# B&R Automation Studio project mappFramework (part 3)

#### AsLoggerFile.c
```c
/********************************************************************
 * COPYRIGHT -- Bernecker + Rainer
 ********************************************************************
 * Library: AsLogger
 * File: AsLoggerFile.c
 * Author: buchananw
 * Created: August 21, 2009
 *******************************************************************/

#include <bur/plctypes.h>
#include <LoggingLib.h>
#include <string.h>
#include <stdbool.h>
#include "AsLoggerInternal.h"

#ifdef __DEBUG_LOGGING_LIBRARY__
#define transit(x, _state)                                          \
{                                                                   \
    x = _state;                                                     \
    logDebug("AsLoggerFile", "changing to state " #_state, NULL);   \
}
#else

#define transit(x, _state)                                          \
{                                                                   \
    x = _state;                                                     \
}

#endif

#define disableAllFunctionBlocks                \
inst->internal.FileOpen_0.enable    = false;    \
inst->internal.FileCreate_0.enable  = false;    \
inst->internal.FileWrite_0.enable   = false;    \
inst->internal.FileCopy_0.enable    = false;    \
inst->internal.FileClose_0.enable   = false;    \
inst->internal.FileDelete_0.enable  = false;

#define incrementFileNumber(x) x = (x+1) % inst->maxFiles
#define decrementFileNumber(x) x = (x > 0) ? x - 1 : inst->maxFiles - 1

void AsLoggerFile(struct AsLoggerFile* inst)
{
    LogStore_typ* logStore;
    UDINT arguments[LOGGING_MAX_ARGUMENTS];
    USINT i;

    if (inst == NULL)
    {
        logError("AsLoggerFile", "AsLoggerFile called with NULL instance", (UDINT)NULL);
        return;
    }
    logStore = getLogStore();

    if (logStore == NULL)
    {
        transit(inst->internal.state, AS_FILE_LOGGER_STATE_ERROR);
#ifdef __DEBUG_LOGGING_LIBRARY__
        logDebug("AsLoggerFile", "logStore is NULL", NULL);
        logDebug("AsLoggerFile", "changing to ERROR state", NULL);
#endif
        inst->status = ASLOGGER_INTERNAL_ERROR;
        return;
    }

    switch(inst->internal.state)
    {
        case AS_FILE_LOGGER_STATE_W_ENABLE:
            if (inst->enable != true)
            {
                inst->status = ERR_FUB_ENABLE_FALSE;
                return;
            }

            if (strcmp(inst->device, "") == true)
            {
                logError("AsLoggerFile", "device name empty", (UDINT)NULL);
                inst->status = ASLOGGER_ILLEGAL_DEVICENAME;
                return;
            }
            if (strcmp(inst->fileName, "") == true)
            {
                logError("AsLoggerFile", "file name empty", (UDINT)NULL);
                inst->status = ASLOGGER_ILLEGAL_FILENAME;
                return;
            }

            inst->internal.fileNumber = (inst->maxFiles > 1) ? inst->maxFiles - 1 : 0;
            if (inst->internal.fileNumber <= 1)
            {
                snprintf2(inst->internal.tempFileName, (sizeof(inst->internal.tempFileName) / sizeof(inst->internal.tempFileName[0])) - 1, "%s.%s", inst->fileName, inst->fileExtension);
                inst->internal.FileDelete_0.pDevice = (UDINT)&inst->device;
                inst->internal.FileDelete_0.pName = (UDINT)&inst->internal.tempFileName;
                inst->internal.FileDelete_0.enable = true;
                transit(inst->internal.state, AS_FILE_LOGGER_STATE_DELETE_OLD);
            }
            else
            {
                snprintf2(inst->internal.newFileName, (sizeof(inst->internal.newFileName) / sizeof(inst->internal.newFileName[0])) - 1, "%s%d.%s", inst->fileName, inst->internal.fileNumber, inst->fileExtension);
                snprintf2(inst->internal.oldFileName, (sizeof(inst->internal.oldFileName) / sizeof(inst->internal.oldFileName[0])) - 1, "%s%d.%s", inst->fileName, --inst->internal.fileNumber, inst->fileExtension);

                inst->internal.FileCopy_0.enable = true;
                inst->internal.FileCopy_0.option = fiOVERWRITE;
                inst->internal.FileCopy_0.pSrc = (UDINT)&inst->internal.oldFileName;
                inst->internal.FileCopy_0.pSrcDev = (UDINT)&inst->device;
                inst->internal.FileCopy_0.pDest = (UDINT)&inst->internal.newFileName;
                inst->internal.FileCopy_0.pDestDev = (UDINT)&inst->device;
                transit(inst->internal.state, AS_FILE_LOGGER_STATE_MOVE_FILES);
            }
        break;

        case AS_FILE_LOGGER_STATE_MOVE_FILES:
            switch (inst->internal.FileCopy_0.status)
            {
                case 0:
                case fiERR_FILE_NOT_FOUND:
                    inst->internal.FileCopy_0.enable = false;
                    if (inst->internal.fileNumber == 0)
                    {
                        snprintf2(inst->internal.tempFileName, (sizeof(inst->internal.tempFileName) / sizeof(inst->internal.tempFileName[0])) - 1, "%s.%s", inst->fileName, inst->fileExtension);
                        inst->internal.FileDelete_0.pDevice = (UDINT)&inst->device;
                        inst->internal.FileDelete_0.pName = (UDINT)&inst->internal.tempFileName;
                        inst->internal.FileDelete_0.enable = true;
                        transit(inst->internal.state, AS_FILE_LOGGER_STATE_DELETE_OLD);
                    }
                    else
                    {
                        strcpy((char*)&inst->internal.newFileName, (char*)&inst->internal.oldFileName);

                        if (inst->internal.fileNumber <= 1)
                        {
                            snprintf2(inst->internal.oldFileName, (sizeof(inst->internal.oldFileName) / sizeof(inst->internal.oldFileName[0])) - 1, "%s.%s", inst->fileName, inst->fileExtension);
                            inst->internal.fileNumber--;
                        }
                        else
                        {
                            snprintf2(inst->internal.oldFileName, (sizeof(inst->internal.oldFileName) / sizeof(inst->internal.oldFileName[0])) - 1, "%s%d.%s", inst->fileName, --inst->internal.fileNumber, inst->fileExtension);
                        }
                        inst->internal.FileCopy_0.option = fiOVERWRITE;
                        inst->internal.FileCopy_0.pSrc = (UDINT)&inst->internal.oldFileName;
                        inst->internal.FileCopy_0.pSrcDev = (UDINT)&inst->device;
                        inst->internal.FileCopy_0.pDest = (UDINT)&inst->internal.newFileName;
                        inst->internal.FileCopy_0.pDestDev = (UDINT)&inst->device;
                        /* no state transition here. */
                    }
                break;

                case ERR_FUB_ENABLE_FALSE:
                    inst->internal.FileCopy_0.enable = true;
                break;

                case ERR_FUB_BUSY:
                break;

                default:
                    disableAllFunctionBlocks;
#ifdef __DEBUG_LOGGING_LIBRARY__
                    //snprintf2(logString, (sizeof(logString) / sizeof(logString[0])) - 1, "old file name %s", inst->internal.oldFileName);
                    //snprintf2(logString, (sizeof(logString) / sizeof(logString[0])) - 1, "new file name %s", inst->internal.newFileName);
                    //logDebug("AsLoggerFile", logString);
                    arguments[0] = (UDINT)inst->internal.oldFileName;
                    arguments[1] = (UDINT)inst->internal.newFileName;
                    logDebug("AsLoggerFile", "old file name is %s, new file name is %s", (UDINT)&arguments);

#endif
                    //snprintf2(logString, (sizeof(logString) / sizeof(logString[0])) - 1, "file copy error %d", inst->internal.FileCopy_0.status);
                    arguments[0] = (UDINT)&inst->internal.FileCopy_0.status;
                    logDebug("AsLoggerFile", "file copy error %d", (UDINT)&arguments);
                    logDebug("AsLoggerFile", "changing to ERROR state", (UDINT)NULL);

                    transit(inst->internal.state, AS_FILE_LOGGER_STATE_ERROR);
                break;
            }
        break;

        case AS_FILE_LOGGER_STATE_DELETE_OLD:

            switch (inst->internal.FileDelete_0.status)
            {
                case 0:
                case fiERR_FILE_NOT_FOUND:
                    inst->internal.FileDelete_0.enable = false;
                    inst->internal.FileCreate_0.pDevice = (UDINT)&inst->device;
                    snprintf2(inst->internal.tempFileName, (sizeof(inst->internal.tempFileName) / sizeof(inst->internal.tempFileName[0]))- 1, "%s.%s", inst->fileName, inst->fileExtension);
                    inst->internal.FileCreate_0.pFile = (UDINT)&inst->internal.tempFileName;
                    inst->internal.FileCreate_0.enable = true;
                    transit(inst->internal.state, AS_FILE_LOGGER_STATE_CREATE_FILE);
                break;

                case ERR_FUB_ENABLE_FALSE:
                    inst->internal.FileDelete_0.enable = true;
                break;

                case ERR_FUB_BUSY:
                break;

                default:
                    disableAllFunctionBlocks;
                    //snprintf2(logString, (sizeof(logString) / sizeof(logString[0])) - 1, "file delete error %d", inst->internal.FileDelete_0.status);
                    arguments[0] = (UDINT)&inst->internal.FileDelete_0.status;
                    logDebug("AsLoggerFile", "file delete error %d", (UDINT)&arguments);
                    logDebug("AsLoggerFile", "changing to ERROR state", (UDINT)NULL);
                    transit(inst->internal.state, AS_FILE_LOGGER_STATE_ERROR);
                break;
            }
        break;

        case AS_FILE_LOGGER_STATE_CREATE_FILE:
            switch (inst->internal.FileCreate_0.status)
            {
                case 0:
                    inst->internal.FileCreate_0.enable = false;
                    inst->internal.FileClose_0.ident = inst->internal.FileCreate_0.ident;
                    inst->internal.FileClose_0.enable = true;
                    inst->internal.fileOffset = 0;
                    inst->internal.writeBufferUsed = 0;
                    transit(inst->internal.state, AS_FILE_LOGGER_STATE_CLOSE);
                break;

                case ERR_FUB_ENABLE_FALSE:
                    inst->internal.FileCreate_0.enable = true;
                break;

                case ERR_FUB_BUSY:
                break;

                default:
                    disableAllFunctionBlocks;
                    //snprintf2(logString, (sizeof(logString) / sizeof(logString[0])) - 1, "file create error %d", inst->internal.FileCreate_0.status);
                    arguments[0] = (UDINT)&inst->internal.FileCreate_0.status;
                    logDebug("AsLoggerFile", "file create error %d", (UDINT)&arguments);
                    logDebug("AsLoggerFile", "changing to ERROR state", (UDINT)NULL);
                    logDebug("AsLoggerFile", inst->internal.tempFileName, (UDINT)NULL);
                    transit(inst->internal.state, AS_FILE_LOGGER_STATE_ERROR);
                    inst->status = inst->internal.FileCreate_0.status;
            }
        break;

        case AS_FILE_LOGGER_STATE_MARSHALL:
            memset(&inst->internal.writeBuffer, 0, sizeof(inst->internal.writeBuffer));
            inst->internal.writeBufferUsed = 0;

            for (i=inst->internal.outputIndex; i != logStore->inputIndex; incrementIndex(i))
            {
                if (logStore->messages[i].level >= inst->level)
                {
                    memset(inst->internal.tempString, 0, sizeof(inst->internal.tempString));
                    marchallLogMessageForFile(&logStore->messages[i], inst->delimiter, inst->internal.tempString, sizeof(inst->internal.tempString) / sizeof(inst->internal.tempString[0]));
                    if ((strlen(inst->internal.tempString) + inst->internal.writeBufferUsed) >= sizeof(inst->internal.writeBuffer))
                    {
                        snprintf2(inst->internal.tempFileName, (sizeof(inst->internal.tempFileName) / sizeof(inst->internal.tempFileName[0])) - 1, "%s.%s", inst->fileName, inst->fileExtension);
                        inst->internal.FileOpen_0.enable = true;
                        inst->internal.FileOpen_0.mode = fiREAD_WRITE;
                        inst->internal.FileOpen_0.pDevice = (UDINT)&inst->device;
                        inst->internal.FileOpen_0.pFile = (UDINT)&inst->internal.tempFileName;
                        transit(inst->internal.state, AS_FILE_LOGGER_STATE_OPEN);
                        return;
                    }
                    addStringToBuffer((char*)&inst->internal.writeBuffer, &inst->internal.writeBufferUsed, inst->internal.tempString);
                }
                incrementIndex(inst->internal.outputIndex);
            }
            if (inst->internal.writeBufferUsed > 0)
            {
                snprintf2(inst->internal.tempFileName, (sizeof(inst->internal.tempFileName) / sizeof(inst->internal.tempFileName[0]))- 1, "%s.%s", inst->fileName, inst->fileExtension);
                inst->internal.FileOpen_0.enable = true;
                inst->internal.FileOpen_0.mode = fiREAD_WRITE;
                inst->internal.FileOpen_0.pDevice = (UDINT)&inst->device;
                inst->internal.FileOpen_0.pFile = (UDINT)&inst->internal.tempFileName;
                transit(inst->internal.state, AS_FILE_LOGGER_STATE_OPEN);
            }
        break;

        case AS_FILE_LOGGER_STATE_OPEN:
            switch (inst->internal.FileOpen_0.status)
            {
                case 0:
                    inst->internal.FileOpen_0.enable = false;

                    inst->internal.FileWrite_0.enable = true;
                    inst->internal.FileWrite_0.ident = inst->internal.FileOpen_0.ident;
                    inst->internal.FileWrite_0.len = inst->internal.writeBufferUsed;
                    inst->internal.FileWrite_0.offset = inst->internal.fileOffset;
                    inst->internal.FileWrite_0.pSrc = (UDINT)inst->internal.writeBuffer;
                    transit(inst->internal.state, AS_FILE_LOGGER_STATE_WRITE);
                break;

                case ERR_FUB_ENABLE_FALSE:
                    inst->internal.FileOpen_0.enable = true;
                break;

                case ERR_FUB_BUSY:
                break;

                default:
                    disableAllFunctionBlocks;
                    //snprintf2(logString, (sizeof(logString) / sizeof(logString[0])) - 1, "file open error %d", inst->internal.FileOpen_0.status);
                    arguments[0] = (UDINT)&inst->internal.FileOpen_0.status;
                    logDebug("AsLoggerFile", "file open error %d", (UDINT)&arguments);
                    logDebug("AsLoggerFile", "changing to ERROR state", (UDINT)NULL);
                    logDebug("AsLoggerFile", inst->internal.tempFileName, (UDINT)NULL);
                    transit(inst->internal.state, AS_FILE_LOGGER_STATE_ERROR);
                    inst->status = inst->internal.FileOpen_0.status;
            }
        break;

        case AS_FILE_LOGGER_STATE_WRITE:
            switch (inst->internal.FileWrite_0.status)
            {
                case 0:
                    inst->internal.FileWrite_0.enable = false;
                    inst->internal.fileOffset += inst->internal.writeBufferUsed;
                    inst->internal.FileClose_0.enable = true;
                    inst->internal.FileClose_0.ident = inst->internal.FileWrite_0.ident;
                    transit(inst->internal.state, AS_FILE_LOGGER_STATE_CLOSE);
                break;

                case ERR_FUB_ENABLE_FALSE:
                    inst->internal.FileWrite_0.enable = true;
                break;

                case ERR_FUB_BUSY:
                break;

                default:
                    disableAllFunctionBlocks;
                    //snprintf2(logString, (sizeof(logString) / sizeof(logString[0])) - 1, "file write error %d", inst->internal.FileWrite_0.status);
                    arguments[0] = (UDINT)&inst->internal.FileWrite_0.status;
                    logDebug("AsLoggerFile", "file write error %d", (UDINT)&arguments);
                    logDebug("AsLoggerFile", "changing to ERROR state", (UDINT)NULL);
                    logDebug("AsLoggerFile", inst->internal.tempFileName, (UDINT)NULL);
                    transit(inst->internal.state, AS_FILE_LOGGER_STATE_ERROR);
                    inst->status = inst->internal.FileWrite_0.status;
            }
        break;

        case AS_FILE_LOGGER_STATE_CLOSE:
            switch (inst->internal.FileClose_0.status)
            {
                case 0:
                    inst->internal.FileClose_0.enable = false;
                    if (inst->internal.fileOffset >= inst->maxFileSize)
                    {
                        inst->internal.fileNumber = (inst->maxFiles > 1) ? inst->maxFiles - 1 : 0;
                        if (inst->internal.fileNumber <= 1)
                        {
                            snprintf2(inst->internal.tempFileName, (sizeof(inst->internal.tempFileName) / sizeof(inst->internal.tempFileName[0])) - 1, "%s.%s", inst->fileName, inst->fileExtension);
                            inst->internal.FileDelete_0.pDevice = (UDINT)&inst->device;
                            inst->internal.FileDelete_0.pName = (UDINT)&inst->internal.tempFileName;
                            inst->internal.FileDelete_0.enable = true;
                            transit(inst->internal.state, AS_FILE_LOGGER_STATE_DELETE_OLD);
                        }
                        else
                        {
                            snprintf2(inst->internal.newFileName, (sizeof(inst->internal.newFileName) / sizeof(inst->internal.newFileName[0])) - 1, "%s%d.%s", inst->fileName, inst->internal.fileNumber, inst->fileExtension);
                            snprintf2(inst->internal.oldFileName, (sizeof(inst->internal.oldFileName) / sizeof(inst->internal.oldFileName[0])) - 1, "%s%d.%s", inst->fileName, --inst->internal.fileNumber, inst->fileExtension);

                            inst->internal.FileCopy_0.enable = true;
                            inst->internal.FileCopy_0.option = fiOVERWRITE;
                            inst->internal.FileCopy_0.pSrc = (UDINT)&inst->internal.oldFileName;
                            inst->internal.FileCopy_0.pSrcDev = (UDINT)&inst->device;
                            inst->internal.FileCopy_0.pDest = (UDINT)&inst->internal.newFileName;
                            inst->internal.FileCopy_0.pDestDev = (UDINT)&inst->device;
                            transit(inst->internal.state, AS_FILE_LOGGER_STATE_MOVE_FILES);
                        }
                    }
                    else
                    {
                        inst->internal.writeBufferUsed = 0;
                        transit(inst->internal.state, AS_FILE_LOGGER_STATE_MARSHALL);
                    }
                break;

                case ERR_FUB_ENABLE_FALSE:
                    inst->internal.FileClose_0.enable = true;
                break;

                case ERR_FUB_BUSY:
                break;

                default:
                    disableAllFunctionBlocks;
                    //snprintf2(logString, (sizeof(logString) / sizeof(logString[0])) - 1, "file close error %d", inst->internal.FileClose_0.status);
                    arguments[0] = (UDINT)&inst->internal.FileClose_0.status;
                    logDebug("AsLoggerFile", "file close error %d", (UDINT)&arguments);
                    logDebug("AsLoggerFile", "changing to ERROR state", (UDINT)NULL);
                    logDebug("AsLoggerFile", inst->internal.tempFileName, (UDINT)NULL);
                    transit(inst->internal.state, AS_FILE_LOGGER_STATE_ERROR);
                    inst->status = inst->internal.FileClose_0.status;
            }
        break;

        case AS_FILE_LOGGER_STATE_ERROR:
            if (inst->enable != true)
            {
                transit(inst->internal.state, 0);
            }
        break;

        default:
        break;
    }

    if (inst->internal.state != AS_FILE_LOGGER_STATE_ERROR)
        inst->status = ERR_FUB_BUSY;

    FileOpen(&inst->internal.FileOpen_0);
    FileWrite(&inst->internal.FileWrite_0);
    FileClose(&inst->internal.FileClose_0);
    FileCreate(&inst->internal.FileCreate_0);
    FileCopy(&inst->internal.FileCopy_0);
    FileDelete(&inst->internal.FileDelete_0);
}

void marchallLogMessageForFile(LogMessage_typ* message, char* delimiter, char* tempString, UDINT sizeOfTempString)
{
    DTStructure timeStamp;
    char level[6];

    if ((message == NULL) || (delimiter == NULL) || (tempString == NULL))
        return;

    DT_TO_DTStructure(message->timeStamp, (UDINT)&timeStamp);
    timeStamp.millisec = message->timeStampMilliseconds;

    memset(&level, 0, sizeof(level));
    switch(message->level)
    {
        case LOG_LEVEL_DEBUG:
            strcpy(level, "DEBUG");
        break;
        case LOG_LEVEL_INFO:
            strcpy(level, "INFO");
        break;
        case LOG_LEVEL_WARN:
            strcpy(level, "WARN");
        break;
        case LOG_LEVEL_ERROR:
            strcpy(level, "ERROR");
        break;
        case LOG_LEVEL_FATAL:
            strcpy(level, "FATAL");
        break;
    }

    snprintf2(tempString, sizeOfTempString - 1, "%04d/%02d/%02d %02d:%02d:%02d.%03d%s %s%s %s%s %s\r\n", timeStamp.year, timeStamp.month, timeStamp.day, \
                    timeStamp.hour, timeStamp.minute, timeStamp.second, timeStamp.millisec, delimiter, \
                    level, delimiter, \
                    message->name, delimiter, \
                    message->message);
}

void addStringToBuffer(char* buffer, UINT* bufferPos, char* newMessage)
{
    if ((buffer == NULL) || (bufferPos == NULL) || (newMessage == NULL))
        return;

    memcpy(buffer + *bufferPos, newMessage, strlen(newMessage));
    *bufferPos = *bufferPos + strlen(newMessage);
}
```

#### AsLoggerLogBook.c
```c
/********************************************************************
 * COPYRIGHT -- Bernecker + Rainer
 ********************************************************************
 * Library: LoggingLib
 * File: AsLoggerLogBook.c
 * Author: buchananw
 * Created: April 19, 2010
 *******************************************************************/

#include <bur/plctypes.h>
#include <LoggingLib.h>
#include <string.h>
#include <stdbool.h>
#include "AsLoggerInternal.h"

#define LOGBOOK_ERROR_STATE 255

#ifdef __DEBUG_LOGGING_LIBRARY__
#define transit(x, y)                                        \
{                                                            \
    x->internal.state = y;                                   \
    logDebug("AsLoggerFile", "changing to state " #y, NULL); \
}
#else
#define transit(x, y)                                        \
{                                                            \
    x->internal.state = y;                                   \
}
#endif

#define incrementFileNumber(x) x = (x+1) % inst->internal.maxFiles
#define decrementFileNumber(x) x = (x > 0) ? x - 1 : inst->internal.maxFiles - 1

void AsLoggerLogBook(struct AsLoggerLogBook* inst)
{
    LogStore_typ* logStore;
#ifdef __DEBUG_LOGGING_LIBRARY__
    UDINT arguments[LOGGING_MAX_ARGUMENTS];
#endif

    if (inst == NULL)
    {
        logError("AsLoggerLogBook", "AsLoggerLogBook called with NULL instance", NULL);
        return;
    }
    logStore = getLogStore();

    if (logStore == NULL)
    {
#ifdef __DEBUG_LOGGING_LIBRARY__
        logDebug("AsLoggerLogBook", "logStore is NULL", NULL);
#endif
        inst->status = ASLOGGER_INTERNAL_ERROR;
        return;
    }

    if (inst->internal.outputIndexRegistered != true)
    {
        addNewOutputIndex(&inst->internal.outputIndex);
        inst->internal.outputIndexRegistered = true;
    }

    while ((inst->internal.outputIndex != logStore->inputIndex) && (logStore->messages[inst->internal.outputIndex].level < inst->level))
    {
        incrementIndex(inst->internal.outputIndex);
    }

    if (inst->internal.outputIndex != logStore->inputIndex)
    {
        if (inst->internal.ArEventLogWrite_0.Ident == 0)
        {
            inst->internal.ArEventLogGetIdent_0.Execute = true;
            strcpy(inst->internal.ArEventLogGetIdent_0.Name, "$arlogusr");
            ArEventLogGetIdent(&inst->internal.ArEventLogGetIdent_0);
            if (inst->internal.ArEventLogGetIdent_0.StatusID == 0)
                inst->internal.ArEventLogWrite_0.Ident = inst->internal.ArEventLogGetIdent_0.Ident;
        }
        else
        {
            USINT _logBuffer[MAX_MESSAGE_LENGTH + MAX_NAME_LENGTH + 10];
            char _tempString[MAX_MESSAGE_LENGTH + MAX_NAME_LENGTH + 2];

            memset(&_logBuffer, 0, sizeof(_logBuffer));
            inst->internal.ArEventLogWrite_0.Execute = true;
            inst->internal.ArEventLogWrite_0.EventID = ArEventLogMakeEventID(convertToArLogLevel(&(logStore->messages[inst->internal.outputIndex])), 0, 0);
            inst->internal.ArEventLogWrite_0.OriginRecordID = 0;
            snprintf2(_tempString, (sizeof(_tempString) / sizeof(_tempString)) - 1, "%s: %s", logStore->messages[inst->internal.outputIndex].name, logStore->messages[inst->internal.outputIndex].message);
            ArEventLogAddDataInit((UDINT)&_logBuffer, sizeof(_logBuffer), arEVENTLOG_ADDFORMAT_CODED);
            ArEventLogAddDataString((UDINT)&_logBuffer, sizeof(_logBuffer), (UDINT)&_tempString);
            inst->internal.ArEventLogWrite_0.AddData = (UDINT)&_logBuffer;
            inst->internal.ArEventLogWrite_0.AddDataFormat = arEVENTLOG_ADDFORMAT_CODED;
            inst->internal.ArEventLogWrite_0.AddDataSize = sizeof(_logBuffer);

            ArEventLogWrite(&inst->internal.ArEventLogWrite_0);
            if (inst->internal.ArEventLogWrite_0.StatusID == 0)
            {
                incrementIndex(inst->internal.outputIndex);

            }
#ifdef __DEBUG_LOGGING_LIBRARY__
            else
            {
                //snprintf2(logString, (sizeof(logString) / sizeof(logString[0])) - 1, "AR log write error %d", inst->internal.AsArLogWrite_0.status);
                arguments[0] = (UDINT)&inst->internal.ArEventLogWrite_0.StatusID;
                logDebug("AsLoggerLogBook", "AR log write error %d", (UDINT)&arguments);
                inst->status = inst->internal.ArEventLogWrite_0.StatusID;
            }
#endif
            inst->internal.ArEventLogWrite_0.Execute = false;
            ArEventLogWrite(&inst->internal.ArEventLogWrite_0);

        }

    }
}

USINT convertToArLogLevel(LogMessage_typ* message)
{
    if (message == NULL)
        return arEVENTLOG_SEVERITY_INFO;

    switch(message->level)
    {
        case LOG_LEVEL_DEBUG:
        case LOG_LEVEL_INFO:
            return arEVENTLOG_SEVERITY_INFO;
        break;
        case LOG_LEVEL_WARN:
            return arEVENTLOG_SEVERITY_WARNING;
        break;
        case LOG_LEVEL_ERROR:
        case LOG_LEVEL_FATAL:
            return arEVENTLOG_SEVERITY_ERROR;
            return arEVENTLOG_SEVERITY_ERROR;
        break;
    }
    return arEVENTLOG_SEVERITY_ERROR;
}
```


### Package Logical/Infrastructure - Package for Machine Infrastructure

### mappFrameworkGlobal.var - Global variables for the mapp Framework
```iecst
(*Recipe*)
VAR CONSTANT
	MACH_CONFIG_CATEGORY_INDEX : USINT := 1; (*Recipe category index for machine config*)
	PARAMETERS_CATEGORY_INDEX : USINT := 0; (*Recipe category index for machine parameters*)
	PARAMETERS_CATEGORY : STRING[10] := 'Parameters'; (*Recipe category for runtime parameters*)
	MACHINE_CONFIGURATION_CATEGORY : STRING[30] := 'Machine Configuration'; (*Recipe category for machine configuration settings*)
	DEFAULT_PARAMETERS : STRING[20] := 'Default'; (*Default parameters recipe file name*)
	PARAMETERS_FILE_EXTENSION : STRING[10] := '.par'; (*File extension for parameter recipe files*)
	DEFAULT_MACHINE_CONFIGURATION : STRING[20] := 'Machine'; (*Default machine configuration recipe file name*)
	MACHINE_CONFIG_FILE_EXTENSION : STRING[10] := '.mcfg'; (*File extension for machine configuration recipe files*)
END_VAR
(*File*)
VAR CONSTANT
	MAX_IDX_USB_DEV_LIST : USINT := 2; (*Maximum number of USB storage devices. Value 2 = 2 USB devices (index 0 and 1)*)
	IDX_USB_DEV_LIST : USINT := MAX_IDX_USB_DEV_LIST - 1; (*Maximum number of USB storage devices.*)
END_VAR
VAR
	gUSBAvailable : ARRAY[0..IDX_USB_DEV_LIST] OF BOOL; (*Boolean array for whether the USB device is plugged in*)
END_VAR
```

### Package Logical/Infrastructure/AlarmX - Package for mapp AlarmX Framework

### Program Logical/Infrastructure/AlarmX/AlarmMgr (IEC) - Alarm manager

#### AlarmMgr.typ
```iecst
(*Structure types*)

TYPE
	AlarmHmiInterfaceType : 	STRUCT  (*Structure to hold commands and status from the HMI*)
		Commands : AlarmCommandsType; (*HMI commands*)
		Status : {REDUND_UNREPLICABLE} AlarmStatusType; (*HMI status*)
		Parameters : AlarmParametersType; (*HMI parameters*)
	END_STRUCT;
	AlarmCommandsType : 	STRUCT  (*Structure to hold the commands from the HMI*)
		ExportAlarms : BOOL; (*Triggers an alarm export of the alarm history. Connected to a button on the HMI.*)
		RunQuery : BOOL; (*Triggers the query to run. Connected to a button on the HMI. *)
	END_STRUCT;
	AlarmParametersType : 	STRUCT  (*Structure to hold the parameters from the HMI*)
		InstanceID : UINT; (*The instanceID of the alarm that was most recently clicked in the AlarmList. Set by an eventbinding in mapp View*)
	END_STRUCT;
	AlarmStatusType : 	STRUCT  (*Structure to hold status information to the mapp View HMI. (This structure is not compatible/relevant if you are using a VC4 visualization)*)
		AlarmHistSortCfg : STRING[1000]; (*Sort configuration property for the AlarmHistory widget *)
		AlarmHistFilterCfg : STRING[1000]; (*Filter configuration property for the AlarmHistory widget*)
		AlarmSortCfg : STRING[1000]; (*Sort configuration for the AlarmList widget*)
		AlarmFilterCfg : STRING[1000]; (*Filter configuration for the AlarmList widget*)
		TableConfig : ARRAY[0..1]OF STRING[120]; (*Table configuration for the alarm query Table*)
		AlarmExportDone : BOOL; (*Alarm export of alarm history is completed. Connected to a button on the HMI. *)
		AlarmExportDisplayed : BOOL; (*Alarm export of alarm history is displayed. Connected to a button on the HMI. *)
		Query : AlarmQueryHMIType; (*Structure which rearranges the query data from AlarmQuery into a structure of arrays for easy connection to the Table widget*)
	END_STRUCT;
	AlarmQueryType : 	STRUCT  (*Structure for query results and status*)
		State : ActiveAlarmStateEnum; (*State variable for the query state machine*)
		LastUpdateCount : UDINT; (*Previous count of query results. Used to check for new query data. *)
		UpdateCount : UDINT; (*Count of query results. Increases each time new results are availble. *)
		Alarms : ARRAY[0..MAX_QUERY_RESULTS]OF AlarmType; (*Query data*)
		Next : BOOL; (*Trigger to query the next data, if there are more results than MAX_QUERY_RESULTS*)
	END_STRUCT;
	AlarmQueryHMIType : 	STRUCT  (*Datatype for the structure which rearranges the query data from AlarmQuery into a structure of arrays for easy connection to the Table widget in mapp View*)
		Active : ARRAY[0..MAX_QUERY_RESULTS]OF BOOL; (*StateActive array*)
		Acknowledged : ARRAY[0..MAX_QUERY_RESULTS]OF BOOL; (*StateAcknowledged array*)
		Scope : ARRAY[0..MAX_QUERY_RESULTS]OF WSTRING[80]; (*Scope array*)
		Name : ARRAY[0..MAX_QUERY_RESULTS]OF STRING[80]; (*Name array*)
		Message : ARRAY[0..MAX_QUERY_RESULTS]OF WSTRING[255]; (*Message array*)
		AdditionalInfo : ARRAY[0..MAX_QUERY_RESULTS]OF WSTRING[255]; (*AdditionalInformation1 array*)
		TimeStamp : ARRAY[0..MAX_QUERY_RESULTS]OF DATE_AND_TIME; (*TimeStamp array*)
		Code : ARRAY[0..MAX_QUERY_RESULTS]OF UDINT; (*Code array*)
		Severity : ARRAY[0..MAX_QUERY_RESULTS]OF UDINT; (*Severity array*)
		State : ARRAY[0..MAX_QUERY_RESULTS]OF CurrentAlarmStateEnum; (*State message array*)
		QueryCount : USINT; (*Count of query results for building the query table configuration string*)
	END_STRUCT;
	AlarmType : 	STRUCT  (*Structure to hold the alarm data for the query results*)
		Active : BOOL; (*ActiveAlarms query, StateActive column*)
		Acknowledged : BOOL; (*ActiveAlarms query, StateAcknowledged column*)
		Scope : WSTRING[80]; (*ActiveAlarms query, Scope column*)
		Name : STRING[80]; (*ActiveAlarms query, Name column*)
		Message : WSTRING[255]; (*ActiveAlarms query, Message column*)
		AdditionalInfo : WSTRING[255]; (*ActiveAlarms query, AdditionalInformation1*)
		TimeStamp : DATE_AND_TIME; (*ActiveAlarms query, TimeStamp column*)
		Code : UDINT; (*ActiveAlarms query, Code column*)
		Severity : UDINT; (*ActiveAlarms query, Severity column*)
		State : CurrentAlarmStateEnum; (*ActiveAlarms query, State column*)
	END_STRUCT;
	MachineDigitalInputsType : 	STRUCT  (*Safety related digital inputs *)
		EmergencyStop : ARRAY[0..MAX_ESTOP]OF BOOL; (*Emergency stop input signals*)
		SafetyDoor : ARRAY[0..MAX_SAFETY_DOOR]OF BOOL; (*Safety door input signals*)
		AcknowledgeAlarms : BOOL; (*Reset button input signal*)
	END_STRUCT;
	AlarmExamplesType : 	STRUCT  (*Structure for alarm samples*)
		LevelMonitoring : INT := 50; (*Triggers LevelMonitoringExample alarm depending on the value set (<20 or >80)*)
		DeviationMonitoring : INT := 15; (*Triggers the DeviationMonitoringExample alarm if this differs from DevationMonitoringSetpoint (below) by more than 5 units*)
		DeviationMonitoringSetpoint : INT := 15; (*Setpoint for the DeviationMonitoringExample alarm. If DeviationMonitoring (above) differs from this value by more than 5 units, the alarm triggers*)
		RateOfChange : INT := 0; (*Triggers the RateOfChangeExample alarm if this value changes at a rate of more than 5 units per second*)
		SnippetValue : INT := 10; (*Process variable used in the SnippetExample alarm for the snippet*)
		SetControlExample : BOOL; (*Boolean to trigger the example alarm which is triggerd by MpAlarmXControlExample_0*)
	END_STRUCT;
END_TYPE

(*Enumerations*)

TYPE
	ActiveAlarmStateEnum :
		( (*Enumeration for the state for the query state machine*)
		ACTIVE_ALARM_WAIT, (*Wait state*)
		ACTIVE_ALARM_QUERY, (*State to query the alarm data*)
		ACTIVE_ALARM_NEXT (*State to check if more alarms meet the query criteria and need to be queried*)
		);
	CurrentAlarmStateEnum :
		( (*Enumeration for the state of a particular alarm*)
		INACTIVE_NOT_ACKNOWLEDGED := 0, (*Alarm inactive and not acknowledged*)
		ACTIVE_NOT_ACKNOWLEDGED := 1, (*Alarm active and not acknowledged*)
		ACTIVE_ACKNOWLEDGED := 2, (*Alarm active and acknowledged*)
		INACTIVE_ACKNOWLEDGED := 3 (*Alarm inactive and acknowledged*)
		);
END_TYPE
```

#### AlarmMgr.var
```iecst
(*Function Blocks*)
VAR
	MpAlarmXHistoryMain : MpAlarmXHistory; (*MpAlarmXHistory instance*)
	MpAlarmXHistoryUIMain : MpAlarmXHistoryUI; (*MpAlarmXHistoryUI instance*)
	MpAlarmXListUIMain : MpAlarmXListUI; (*MpAlarmXList instance*)
	MpAlarmXCoreMain : MpAlarmXCore; (*MpAlarmXCore instance*) (*ChangeStyleAlarmButton : USINT := 0; (*changeStyle of a AlarmFlyout in mappView*)
	MpAlarmXControlExample : {REDUND_UNREPLICABLE} MpAlarmXAlarmControl; (*MpAlarmXAlarmControl instance*)
	QueryActiveAlarms : {REDUND_UNREPLICABLE} MpAlarmXQuery; (*MpAlarmXQuery instance*)
	DirCreateAlarm : DirCreate; (*DirCreate instance*)
END_VAR
(*Constants*)
VAR CONSTANT
	MAX_QUERY_RESULTS : USINT := 19; (*Maximum number of query results (Value+1)*)
	MAX_SAFETY_DOOR : UINT := 5; (*Maximum number of safety doors (Value+1)*)
	MAX_ESTOP : UINT := 2; (*Maximum number of emergency stops (Value+1)*)
END_VAR
(*Structure Types*)
VAR
	HmiAlarmX : AlarmHmiInterfaceType; (*HMI interface structure*)
	MpAlarmXListUIConnect : MpAlarmXListUIConnectType := (0); (*AlarmX list connection to the UI*)
	MpAlarmXHistoryUIConnect : MpAlarmXHistoryUIConnectType; (*AlarmX History connection to the UI*)
	SafetyInputs : MachineDigitalInputsType; (*Safety related digital inputs*)
	AlarmExamples : {REDUND_UNREPLICABLE} AlarmExamplesType; (*Sample alarms for different monitoring types*)
	AlarmQuery : {REDUND_UNREPLICABLE} AlarmQueryType; (*Query results and status*)
END_VAR
(*Variables*)
VAR
	Alarms : {REDUND_UNREPLICABLE} ARRAY[0..99] OF BOOL; (*Array of monitored alarm bits*)
	CommissioningModeActive : {REDUND_UNREPLICABLE} BOOL; (*Boolean value to enable commissioning mode. By default, this inhibits the Alarms[0] alarm*)
	i : USINT; (*Index for loops*)
	MaxIndex : USINT; (*Maximum index for the alarm list*)
END_VAR
```

#### AlarmHandling.st
```iecst
ACTION AlarmHandling:

    // CommissioningModeActive = TRUE will inhibit Alarms[0]. The alarm will not trigger even if the alarm condition is active.
    // CommissioningModeActive = FALSE will NOT inhibit Alarms[0]. The alarm will trigger when the alarm condition is active.
    // See Alarm.mpalarmxcore (must enable Advanced Features)
    CommissioningModeActive;

    // Define the condition which triggers each alarm below.
    Alarms[0];

//	Alarms[1] := ;
//	Alarms[2] := ;
//	Alarms[3] := ;
//	Alarms[4] := ;
//	Alarms[5] := ;
//	Alarms[6] := ;
//	Alarms[7] := ;
//	Alarms[8] := ;
//	Alarms[9] := ;
//
//	Alarms[10] := ;
//	Alarms[11] := ;
//	Alarms[12] := ;
//	Alarms[13] := ;
//	Alarms[14] := ;
//	Alarms[15] := ;
//	Alarms[16] := ;
//	Alarms[17] := ;
//	Alarms[18] := ;
//	Alarms[19] := ;
//
//	Alarms[20] := ;
//	Alarms[21] := ;
//	Alarms[22] := ;
//	Alarms[23] := ;
//	Alarms[24] := ;
//	Alarms[25] := ;
//	Alarms[26] := ;
//	Alarms[27] := ;
//	Alarms[28] := ;
//	Alarms[29] := ;
//
//	Alarms[30] := ;
//	Alarms[31] := ;
//	Alarms[32] := ;
//	Alarms[33] := ;
//	Alarms[34] := ;
//	Alarms[35] := ;
//	Alarms[36] := ;
//	Alarms[37] := ;
//	Alarms[38] := ;
//	Alarms[39] := ;
//
//	Alarms[40] := ;
//	Alarms[41] := ;
//	Alarms[42] := ;
//	Alarms[43] := ;
//	Alarms[44] := ;
//	Alarms[45] := ;
//	Alarms[46] := ;
//	Alarms[47] := ;
//	Alarms[48] := ;
//	Alarms[49] := ;
//
//	Alarms[50] := ;
//	Alarms[51] := ;
//	Alarms[52] := ;
//	Alarms[53] := ;
//	Alarms[54] := ;
//	Alarms[55] := ;
//	Alarms[56] := ;
//	Alarms[57] := ;
//	Alarms[58] := ;
//	Alarms[59] := ;
//
//	Alarms[60] := ;
//	Alarms[61] := ;
//	Alarms[62] := ;
//	Alarms[63] := ;
//	Alarms[64] := ;
//	Alarms[65] := ;
//	Alarms[66] := ;
//	Alarms[67] := ;
//	Alarms[68] := ;
//	Alarms[69] := ;
//
//	Alarms[70] := ;
//	Alarms[71] := ;
//	Alarms[72] := ;
//	Alarms[73] := ;
//	Alarms[74] := ;
//	Alarms[75] := ;
//	Alarms[76] := ;
//	Alarms[77] := ;
//	Alarms[78] := ;
//	Alarms[79] := ;
//
//	Alarms[80] := ;
//	Alarms[81] := ;
//	Alarms[82] := ;
//	Alarms[83] := ;
//	Alarms[84] := ;
//	Alarms[85] := ;
//	Alarms[86] := ;
//	Alarms[87] := ;
//	Alarms[88] := ;
//	Alarms[89] := ;
//
//	Alarms[90] := ;
//	Alarms[91] := ;
//	Alarms[92] := ;
//	Alarms[93] := ;
//	Alarms[94] := ;
//	Alarms[95] := ;
//	Alarms[96] := ;
//	Alarms[97] := ;
//	Alarms[98] := ;
//	Alarms[99] := ;

END_ACTION
```

#### AlarmMgr.st
```iecst
//***********************************************************************
// Copyright: B&R Industrial Automation GmbH
// Author: B&R Industrial Automation GmbH
// Created: April 12, 2022
// Description: Tasks for alarm management.
//***********************************************************************

PROGRAM _INIT

	// Create folder for this component on the user file device
	DirCreate_0(enable := TRUE, pDevice := ADR('mappAlarmXFiles'), pName := ADR('/'));

	// Check if folder already exist and if so disabled the function block call
	IF DirCreate_0.status = fiERR_DIR_ALREADY_EXIST THEN
		DirCreate_0(enable := FALSE);
	END_IF

	// Call action to intialize alarm samples
	AlarmSampleInit;

	// Initialize mapp function blocks
	MpAlarmXCore_0.Enable := TRUE;
	MpAlarmXCore_0.MpLink := ADR(gMpLinkAlarmXCore);
	MpAlarmXCore_0();

	MpAlarmXHistory_0.Enable := TRUE;
	MpAlarmXHistory_0.DeviceName := ADR('mappAlarmXFiles');
	MpAlarmXHistory_0.MpLink := ADR(gMpLinkAlarmXHistory);
	MpAlarmXHistory_0();

	MpAlarmXListUI_0.Enable := TRUE;
	MpAlarmXListUI_0.MpLink := ADR(gMpLinkAlarmXCore);
	MpAlarmXListUI_0.UISetup.AlarmListScrollWindow := 10;
	MpAlarmXListUI_0.UISetup.AlarmListSize := 50;
	MpAlarmXListUI_0.UISetup.TimeStampPattern := '%Y %m %d %H:%M:%S';
	MpAlarmXListUI_0();

	MpAlarmXHistoryUI_0.Enable := TRUE;
	MpAlarmXHistoryUI_0.MpLink := ADR(gMpLinkAlarmXHistory);
	MpAlarmXHistoryUI_0.UISetup.AlarmListScrollWindow := 10;
	MpAlarmXHistoryUI_0.UISetup.AlarmListSize := (SIZEOF(MpAlarmXListUIConnect.AlarmList.InstanceID) / SIZEOF(MpAlarmXListUIConnect.AlarmList.InstanceID[0]));
	MpAlarmXHistoryUI_0.UISetup.TimeStampPattern := '%Y %m %d %H:%M:%S';
	MpAlarmXHistoryUI_0();

END_PROGRAM

PROGRAM _CYCLIC

	IF EDGEPOS(SafetyInputs.AcknowledgeAlarms) THEN
		MpAlarmXListUIConnect.AcknowledgeAll := TRUE;
	END_IF

	// Call all cyclic actions
	AlarmHandling;
	GetBacktraceInformation;
	ExecuteQuery;
	QueryTableConfig;
	AlarmSampleFub;
	ExportAlarms;

	// Check if any reactions are active.
	// Typically the MpAlarmXCheckReaction() function is called from other tasks within the application.
	// For example, the axis control task might check for the 'Error' reaction to determine whether to send a stop command to the axes.
	// Therefore, copy/paste these IF statements to other places in the application as needed.
	IF MpAlarmXCheckReaction(gMpLinkAlarmXCore, 'Error') THEN
		// Error is active. Add code here to respond to error situation.
	ELSIF MpAlarmXCheckReaction(gMpLinkAlarmXCore, 'Warning') THEN
		// Warning is active. Add code here to respond to warning situation.
	ELSIF MpAlarmXCheckReaction(gMpLinkAlarmXCore, 'Info') THEN
		// Info is active. Add code here to resond to info situation.
	END_IF

	// Error reset
	IF NOT MpAlarmXCore_0.Error THEN
		MpAlarmXCore_0.ErrorReset := FALSE;
	END_IF
	IF NOT MpAlarmXListUI_0.Error THEN
		MpAlarmXListUI_0.ErrorReset := FALSE;
	END_IF
	IF NOT MpAlarmXHistory_0.Error THEN
		MpAlarmXHistory_0.ErrorReset := FALSE;
	END_IF
	IF NOT MpAlarmXHistoryUI_0.Error THEN
		MpAlarmXHistoryUI_0.ErrorReset := FALSE;
	END_IF

	// Assign MpLinks & address references
	MpAlarmXCore_0.MpLink := ADR(gMpLinkAlarmXCore);
	MpAlarmXListUI_0.MpLink := ADR(gMpLinkAlarmXCore);
	MpAlarmXListUI_0.UIConnect := ADR(MpAlarmXListUIConnect);
	MpAlarmXHistory_0.MpLink := ADR(gMpLinkAlarmXHistory);
	MpAlarmXHistory_0.DeviceName := ADR('mappAlarmXFiles');
	MpAlarmXHistoryUI_0.MpLink := ADR(gMpLinkAlarmXHistory);
	MpAlarmXHistoryUI_0.UIConnect := ADR(MpAlarmXHistoryUIConnect);

	// Call function blocks
	MpAlarmXCore_0();
	MpAlarmXListUI_0();
	MpAlarmXHistory_0();
	MpAlarmXHistoryUI_0();

END_PROGRAM

PROGRAM _EXIT

	// Disable the function blocls to unlink the MpLinks
	MpAlarmXCore_0.Enable := FALSE;
	MpAlarmXListUI_0.Enable := FALSE;
	MpAlarmXHistory_0.Enable := FALSE;
	MpAlarmXHistoryUI_0.Enable := FALSE;
	QueryActiveAlarms_0.Enable := FALSE;

	// Call function blocks
	MpAlarmXCore_0();
	MpAlarmXListUI_0();
	MpAlarmXHistory_0();
	MpAlarmXHistoryUI_0();
	QueryActiveAlarms_0();

END_PROGRAM
```

#### AlarmSamples.st
```iecst
ACTION AlarmSampleInit:

	// Call all variables that are needed for the alarm examples and explain all examples in comments

	// If AlarmExamples.LevelMonitoring gets less than 20 or more than 80, the LevelMonitoringExample alarm will trigger
	// The Low limit is 20. The LowLow limit is 10. The High limit is 80. The HighHigh limit is 90.
	AlarmExamples.LevelMonitoring := 50;

	// If AlarmExamples.DeviationMonitoring deviates from the setpoint (AlarmExamples.DeviationMonitoringSetpoint) by more than 5
	// units in either direction, the DeviationMonitoringExample alarm will trigger
	AlarmExamples.DeviationMonitoring := 15;
	AlarmExamples.DeviationMonitoringSetpoint := 15;

	// If AlarmExamples.RateOfChange increases at a rate of more than 5 units per second, the RateOfChangeExample alarm will trigger
	AlarmExamples.RateOfChange := 0;

	// If AlarmExamples.SnippetValue gets between 50 and 100, an alarm will trigger and the current value will be shown in the alarm text
	AlarmExamples.SnippetValue := 10;

END_ACTION

ACTION AlarmSampleFub:

	// Example of using the MpAlarmXControl() function block.
	// Typically this function is called from other tasks within the application (decentralized).
	// For example, if you have an error in the recipe system, you can trigger it directly in the recipe task.
	// Therefore, copy/paste this example to other places in the application as needed.
	MpAlarmXControlExample.MpLink := ADR(gMpLinkAlarmXCore);
	MpAlarmXControlExample.Enable := TRUE;
	MpAlarmXControlExample.Name := ADR('MpAlarmXControlExample');
	MpAlarmXControlExample.Set := AlarmExamples.SetControlExample;
	MpAlarmXControlExample();

END_ACTION
```

#### ExecuteQuery.st
```iecst
ACTION ExecuteQuery:

	// Initialize mapp function block
	QueryActiveAlarms.MpLink := ADR(gMpLinkAlarmXCore);
	QueryActiveAlarms.Enable := TRUE;
	QueryActiveAlarms.Name := ADR('ActiveAlarms');
	QueryActiveAlarms.Language := ADR('en');
	QueryActiveAlarms();

	CASE (AlarmQuery.State) OF
		ACTIVE_ALARM_WAIT:
			// Wait until the RunQuery command is triggered from the HMI.
			// If you prefer that the query runs anytime new data is available, then uncomment line 15 and comment out line 16 and delete
			// the "Run query" button from the HMI.
			//IF (AlarmQuery.LastUpdateCount <> AlarmQuery.UpdateCount) THEN
			IF (HmiAlarmX.Commands.RunQuery) THEN
				brsmemset(ADR(AlarmQuery.Alarms[0]), 0, SIZEOF(AlarmQuery.Alarms));
				AlarmQuery.LastUpdateCount := AlarmQuery.UpdateCount;
				QueryActiveAlarms.Execute := TRUE;
				HmiAlarmX.Commands.RunQuery := FALSE;
				AlarmQuery.State := ACTIVE_ALARM_QUERY;
			END_IF

		ACTIVE_ALARM_QUERY:
			// If the number of query results is less than MAX_QUERY_RESULTS, return to the wait state
			IF (QueryActiveAlarms.CommandDone AND (NOT QueryActiveAlarms.Info.HasMoreRows)) THEN
				QueryActiveAlarms.Execute := FALSE;
				QueryActiveAlarms.Next := FALSE;
				AlarmQuery.State := ACTIVE_ALARM_WAIT;
				// If the number of query results is more than MAX_QUERY_RESULTS, then query the next set of results
			ELSIF ((QueryActiveAlarms.CommandDone) AND (QueryActiveAlarms.Info.HasMoreRows)) THEN
				QueryActiveAlarms.Next := FALSE;
				AlarmQuery.State := ACTIVE_ALARM_NEXT;
			END_IF

		ACTIVE_ALARM_NEXT:
			IF (AlarmQuery.Next) THEN
				// By default, AlarmQuery.Alarms has 20 elements, so it can hold 20 query results at a time (MAX_QUERY_RESULTS = 19).
				// If AlarmQuery.Next is true, this means the query result is more than 20 alarms.
				// If you want to save the data for the first 20 alarms, add code here to copy AlarmQuery.Alarms to another location.
				// Otherwise, the older alarms in the query will get overwritten with the newest entries here.
				brsmemset(ADR(AlarmQuery.Alarms[0]), 0, SIZEOF(AlarmQuery.Alarms));
				AlarmQuery.Next := FALSE;
				QueryActiveAlarms.Next := TRUE;
				AlarmQuery.State := ACTIVE_ALARM_QUERY;
			END_IF
	END_CASE

	// Convert the query results into arrays that can easily be bound to the Table widget in mapp View
	FOR i := 0 TO MAX_QUERY_RESULTS DO
		HmiAlarmX.Status.Query.Active[i] := AlarmQuery.Alarms[i].Active;
		HmiAlarmX.Status.Query.Acknowledged[i] := AlarmQuery.Alarms[i].Acknowledged;
		HmiAlarmX.Status.Query.Scope[i] := AlarmQuery.Alarms[i].Scope;
		HmiAlarmX.Status.Query.Name[i] := AlarmQuery.Alarms[i].Name;
		HmiAlarmX.Status.Query.Message[i] := AlarmQuery.Alarms[i].Message;
		HmiAlarmX.Status.Query.AdditionalInfo[i] := AlarmQuery.Alarms[i].AdditionalInfo;
		HmiAlarmX.Status.Query.TimeStamp[i] := AlarmQuery.Alarms[i].TimeStamp;
		HmiAlarmX.Status.Query.Severity[i] := AlarmQuery.Alarms[i].Severity;

		IF HmiAlarmX.Status.Query.Active[i] AND NOT HmiAlarmX.Status.Query.Acknowledged[i] THEN
			HmiAlarmX.Status.Query.State[i] := ACTIVE_NOT_ACKNOWLEDGED;
		ELSIF HmiAlarmX.Status.Query.Active[i] AND HmiAlarmX.Status.Query.Acknowledged[i] THEN
			HmiAlarmX.Status.Query.State[i] := ACTIVE_ACKNOWLEDGED;
		ELSIF NOT HmiAlarmX.Status.Query.Active[i] AND NOT HmiAlarmX.Status.Query.Acknowledged[i] THEN
				HmiAlarmX.Status.Query.State[i] := INACTIVE_NOT_ACKNOWLEDGED;
		ELSIF NOT HmiAlarmX.Status.Query.Active[i] AND HmiAlarmX.Status.Query.Acknowledged[i] THEN
				HmiAlarmX.Status.Query.State[i] := INACTIVE_ACKNOWLEDGED;
		END_IF

	END_FOR

END_ACTION
```

#### HMIActions.st
```iecst
ACTION GetBacktraceInformation:

	MaxIndex := (SIZEOF(MpAlarmXListUIConnect.AlarmList.InstanceID)/SIZEOF(MpAlarmXListUIConnect.AlarmList.InstanceID[0])) - 1;
	// Find selected alarm in order to show backtrace information
	FOR i := 0 TO MaxIndex DO
		IF (MpAlarmXCoreMain.PendingAlarms = 0) THEN
			// No pending alarms, reset instance id
			HmiAlarmX.Parameters.InstanceID := 0;
			EXIT;
		END_IF

		IF (MpAlarmXListUIConnect.AlarmList.InstanceID[i] = HmiAlarmX.Parameters.InstanceID) THEN
			// Found an alarm
			MpAlarmXListUIConnect.AlarmList.SelectedIndex := i;
			EXIT;
		END_IF

		IF (MpAlarmXListUIConnect.AlarmList.InstanceID[i] = 0) THEN
			IF (MpAlarmXCoreMain.PendingAlarms > i) THEN
				// Alarm not found, list can page up
				MpAlarmXListUIConnect.AlarmList.PageUp := TRUE;
			END_IF
			EXIT;
		ELSIF (i = MaxIndex) THEN
			// Alarm not found, list can page down
			MpAlarmXListUIConnect.AlarmList.PageDown := TRUE;
		END_IF
	END_FOR

END_ACTION

ACTION QueryTableConfig:

	// Configure visible list
	HmiAlarmX.Status.TableConfig[0] := '{ "specRows": [{"from":';
	HmiAlarmX.Status.Query.QueryCount := 0;
	FOR i := 0 TO 9 DO
		IF HmiAlarmX.Status.Query.Message[i] <> "" THEN
			HmiAlarmX.Status.Query.QueryCount := i + 1;
		END_IF
	END_FOR
	brsitoa((HmiAlarmX.Status.Query.QueryCount), ADR(HmiAlarmX.Status.TableConfig[0]) + brsstrlen(ADR(HmiAlarmX.Status.TableConfig[0])));
	brsstrcat(ADR(HmiAlarmX.Status.TableConfig[0]), ADR(',"to":19, "visible":false}]}'));

END_ACTION

ACTION ExportAlarms:

	IF (HmiAlarmX.Commands.ExportAlarms) THEN
		MpAlarmXHistoryMain.Export := TRUE;
	END_IF

	IF ((MpAlarmXHistoryMain.Export) AND (MpAlarmXHistoryMain.CommandDone)) THEN
		MpAlarmXHistoryMain.Export := FALSE;
		HmiAlarmX.Commands.ExportAlarms := FALSE;
		HmiAlarmX.Status.AlarmExportDone := TRUE;
	END_IF

	IF HmiAlarmX.Status.AlarmExportDisplayed THEN
		HmiAlarmX.Status.AlarmExportDisplayed := FALSE;
		HmiAlarmX.Status.AlarmExportDone := FALSE;
	END_IF

END_ACTION
```

- AlarmImportExport.py - Python script to Import or Export mpAlarmXCore files (not shown)

- test_AlarmImportExport.py - Unit Tests for AlarmImportExport (not shown)

### Package Logical/Infrastructure/Backup - Package for mapp Backup Framework

### Program Logical/Infrastructure/Backup/BackupMgr (IEC)

#### BackupMgr.st - Init, cyclic, exit code
```iecst
//***********************************************************************
// Copyright: B&R Industrial Automation GmbH
// Author: B&R Industrial Automation GmbH
// Created: April 12, 2022
// Description: Task for backup management.
//***********************************************************************

PROGRAM _INIT

	// Create folder for this component on the user file device
	DirCreateBackup(enable := TRUE, pDevice := ADR('mappBackupFiles'), pName := ADR('/'));

	// Check if folder already exist and if so disabled the function block call
	IF DirCreateBackup.status = fiERR_DIR_ALREADY_EXIST THEN
		DirCreateBackup(enable := FALSE);
	END_IF

	// Initialize mapp function blocks
	MpBackupCoreSys.MpLink := ADR(gMpLinkBackupCore);
	MpBackupCoreSys.Enable := TRUE;
	MpBackupCoreSys();

	MpFileManagerUIBackup.UISetup.FileListSize := 50;
	FOR i:=0 TO ((SIZEOF(MpFileManagerUIConnect.DeviceList.DeviceNames)/SIZEOF(MpFileManagerUIConnect.DeviceList.DeviceNames[0])) - 1) DO
		MpFileManagerUIConnect.DeviceList.DeviceNames[i] := '';
	END_FOR
	MpFileManagerUIConnect.DeviceList.DeviceNames[0] := 'mappBackupFiles';

	MpFileManagerUIBackup.MpLink := ADR(gMpLinkFileManagerUIBackup);
	MpFileManagerUIBackup.UIConnect := ADR(MpFileManagerUIConnect);
	MpFileManagerUIBackup.Enable := TRUE;
	MpFileManagerUIBackup();

	MpBackupCoreConfigSys.Enable := TRUE;
	MpBackupCoreConfigSys.MpLink := ADR(gMpLinkBackupCore);
	MpBackupCoreConfigSys.Configuration := ADR(MpBackupConfiguration);

	MpBackupCoreConfigSys.Load := NOT(DiagCpuIsARsim() OR DiagCpuIsSimulated());

	MpBackupCoreConfigSys();

	HmiBackup.Status.DeviceDataProvider[0] := '{"value":"mappBackupFiles","text":"CF/PLC"}';

	// Restored the retained values to the backup settings
	HmiBackup.Parameters.AutomaticBackup := AutomaticBackupRetain;

END_PROGRAM

PROGRAM _CYCLIC

	// Call all cyclic actions
	FileManager;
	IF NOT DiagCpuIsARsim() THEN
		ChangeConfiguration;
	END_IF
	FormatDeviceDataProvider;

	CASE BackupState OF
		BACKUP_IDLE:
			HmiBackup.Status.CreateAllowed := NOT(MpBackupCoreSys.Info.Automatic.Backup.InProgress) AND NOT HmiBackup.Status.SimulationActive;
			HmiBackup.Status.Busy := FALSE;
			IF (MpBackupCoreSys.Error) THEN
				MpBackupCoreSys.ErrorReset := FALSE;
				BackupState := BACKUP_ERROR;
			ELSIF DiagCpuIsARsim() OR DiagCpuIsSimulated() THEN
				HmiBackup.Status.CreateAllowed := FALSE;
				HmiBackup.Status.RestoreAllowed := FALSE;
				BackupState := BACKUP_SIM;
			ELSIF (HmiBackup.Commands.Create) THEN
				HmiBackup.Commands.Create := FALSE;
				MpBackupCoreSys.Create := TRUE;
				HmiBackup.Status.Busy := TRUE;
				HmiBackup.Status.CreateAllowed := FALSE;
				HmiBackup.Status.RestoreAllowed := FALSE;
				MpBackupCoreSys.Name := ADR(HmiBackup.Parameters.Name);
				BackupState := BACKUP_CREATING;
			ELSIF MpBackupCoreSys.Info.Automatic.Backup.InProgress THEN
				HmiBackup.Status.Busy := TRUE;
				HmiBackup.Status.CreateAllowed := FALSE;
				HmiBackup.Status.RestoreAllowed := FALSE;
				BackupState := BACKUP_AUTOCREATE;
			ELSIF (HmiBackup.Commands.Restore) THEN
				HmiBackup.Commands.Restore := FALSE;
				MpBackupCoreSys.Install := TRUE;
				HmiBackup.Status.Busy := TRUE;
				HmiBackup.Status.CreateAllowed := FALSE;
				HmiBackup.Status.RestoreAllowed := FALSE;
				MpBackupCoreSys.Name := ADR(MpFileManagerUIConnect.File.List.Items[HmiBackup.Status.SelectedIndex].Name);
				BackupState := BACKUP_RESTORING;
			ELSIF (HmiBackup.Commands.Update) THEN
				HmiBackup.Commands.Update := FALSE;
				MpBackupCoreSys.Install := TRUE;
				HmiBackup.Status.Busy := TRUE;
				HmiBackup.Status.CreateAllowed := FALSE;
				HmiBackup.Status.RestoreAllowed := FALSE;
				MpBackupCoreSys.Name := ADR(MpBackupCoreSys.Info.Automatic.Update.Name);
				BackupState := BACKUP_UPDATING;
			ELSIF (HmiBackup.Commands.Delete) THEN
				MpFileManagerUIConnect.File.List.Items[HmiBackup.Status.SelectedIndex].IsSelected := TRUE;
				HmiBackup.Commands.Delete := FALSE;
				MpFileManagerUIConnect.File.Delete := TRUE;
				BackupState := BACKUP_DELETING;
			ELSIF (HmiBackup.Commands.SaveConfig) THEN
				HmiBackup.Commands.SaveConfig := FALSE;
				SaveBackupConfiguration;
				MpBackupCoreConfigSys.Save := TRUE;
			ELSIF ((HmiBackup.Status.SelectedIndex <> HmiBackup.Status.LastSelectedIndex) AND (MpBackupCoreSys.CommandBusy <> TRUE)) THEN
				HmiBackup.Status.LastSelectedIndex := HmiBackup.Status.SelectedIndex;
				MpBackupCoreSys.Name := ADR(MpFileManagerUIConnect.File.List.Items[HmiBackup.Status.SelectedIndex].Name);
				IF MpFileManagerUIConnect.File.List.Items[HmiBackup.Status.SelectedIndex].Name <> '' THEN
					MpBackupCoreSys.RequestInfo := TRUE;
				END_IF
			END_IF

		BACKUP_CREATING:
			IF (MpBackupCoreSys.CommandDone) THEN
				MpBackupCoreSys.Create := FALSE;
				MpBackupCoreSys.Install := FALSE;
				MpBackupCoreSys.RequestInfo := FALSE;
				MpFileManagerUIConnect.File.Refresh := TRUE;
				BackupState := BACKUP_REFRESHING_LIST;
			ELSIF (MpBackupCoreSys.Error) THEN
				BackupState := BACKUP_ERROR;
			END_IF

		BACKUP_AUTOCREATE:
			IF NOT MpBackupCoreSys.Info.Automatic.Backup.InProgress THEN
				MpBackupCoreSys.Install := FALSE;
				MpBackupCoreSys.RequestInfo := FALSE;
				MpFileManagerUIConnect.File.Refresh := TRUE;
				BackupState := BACKUP_REFRESHING_LIST;
			ELSIF (MpBackupCoreSys.Error) THEN
				BackupState := BACKUP_ERROR;
			END_IF

		BACKUP_REFRESHING_LIST:
			IF MpFileManagerUIConnect.Status = mpFILE_UI_STATUS_REFRESH THEN
				// Wait for the list to be refreshed with the newly created backup file
			ELSIF MpFileManagerUIConnect.Status = mpFILE_UI_STATUS_IDLE THEN
				HmiBackup.Status.LastSelectedIndex := HmiBackup.Status.LastSelectedIndex + 1;
				BackupState := BACKUP_IDLE;
			ELSIF (MpBackupCoreSys.Error) THEN
				BackupState := BACKUP_ERROR;
			END_IF

		BACKUP_RESTORING:
			IF (MpBackupCoreSys.CommandDone) THEN
				MpBackupCoreSys.Create := FALSE;
				MpBackupCoreSys.Install := FALSE;
				MpBackupCoreSys.RequestInfo := FALSE;
				MpFileManagerUIConnect.File.Refresh := TRUE;
				BackupState := BACKUP_IDLE;
			ELSIF (MpBackupCoreSys.Error) THEN
				BackupState := BACKUP_ERROR;
			END_IF

		BACKUP_UPDATING:
			IF (MpBackupCoreSys.CommandDone) THEN
				MpBackupCoreSys.Create := FALSE;
				MpBackupCoreSys.Install := FALSE;
				MpBackupCoreSys.RequestInfo := FALSE;
				BackupState := BACKUP_IDLE;
			ELSIF (MpBackupCoreSys.Error) THEN
				BackupState := BACKUP_ERROR;
			END_IF

		BACKUP_DELETING:
			CASE (MpFileManagerUIConnect.MessageBox.Type) OF
				mpFILE_MSG_CONFIRM_DELETE:
					MpFileManagerUIConnect.MessageBox.Confirm := TRUE;
				mpFILE_MSG_OK:
					IF (MpFileManagerUIConnect.Status = mpFILE_UI_STATUS_IDLE) THEN
						HmiBackup.Status.LastSelectedIndex := HmiBackup.Status.LastSelectedIndex + 1;
						FOR i := 0 TO ((SIZEOF(MpFileManagerUIConnect.File.List.Items[i])/SIZEOF(MpFileManagerUIConnect.File.List.Items[0])) - 1) DO
							MpFileManagerUIConnect.File.List.Items[i].IsSelected := FALSE;
						END_FOR
						HmiBackup.Status.SelectedIndex := 0;
						MpFileManagerUIConnect.MessageBox.Confirm := FALSE;
						BackupState := BACKUP_IDLE;
					END_IF
			END_CASE

		BACKUP_SIM:
			HmiBackup.Status.SimulationActive := TRUE;

		BACKUP_ERROR:
			MpBackupCoreSys.Create := FALSE;
			MpBackupCoreSys.Install := FALSE;
			IF MpBackupCoreSys.Info.Diag.StatusID.ID <> 0 THEN //-1064159486
				HmiBackup.Status.Error := TRUE;
			END_IF
			IF HmiBackup.Commands.Reset OR (MpBackupCoreSys.Info.Diag.StatusID.ID = -1064159486) THEN
				HmiBackup.Commands.Reset := FALSE;
				MpBackupCoreSys.ErrorReset := TRUE;
				BackupState := BACKUP_IDLE;
			ELSIF ((MpBackupCoreSys.Info.Diag.StatusID.ID = 0) AND (NOT MpBackupCoreSys.Error)) THEN
				BackupState := BACKUP_IDLE;
			END_IF
	END_CASE

	// Reset any errors caused by requesting information
	IF EDGEPOS((MpBackupCoreSys.Error) AND (MpBackupCoreSys.RequestInfo)) THEN
		MpBackupCoreSys.ErrorReset := TRUE;
		MpBackupCoreSys.RequestInfo := FALSE;
		brsmemset(ADR(HmiBackup.Status.Info), 0, SIZEOF(HmiBackup.Status.Info));
	END_IF

	MpBackupCoreSys.MpLink := ADR(gMpLinkBackupCore);
	MpBackupCoreSys.DeviceName := ADR(MpFileManagerUIConnect.DeviceList.DeviceNames[MpFileManagerUIConnect.DeviceList.SelectedIndex]);
	MpBackupCoreSys();

	IF (MpBackupCoreSys.CommandDone) AND (MpBackupCoreSys.RequestInfo) THEN
		MpBackupCoreSys.RequestInfo := FALSE;
		HmiBackup.Status.Info := MpBackupCoreSys.Info.Project.Requested;
	END_IF
	IF EDGEPOS(NOT MpBackupCoreSys.Error) THEN
		MpBackupCoreSys.ErrorReset := FALSE;
		HmiBackup.Status.Error := FALSE;
	END_IF

	HmiBackup.Status.RestoreAllowed := (MpFileManagerUIConnect.File.PathInfo.FolderCount > 0) AND NOT(MpBackupCoreSys.Info.Automatic.Backup.InProgress) AND NOT HmiBackup.Status.SimulationActive;
	HmiBackup.Status.Update := MpBackupCoreSys.Info.Automatic.Update;
	HmiBackup.Status.BackupCtrlEnabled := (NOT HmiBackup.Status.SimulationActive);

	// Assign MpLinks & address references
	MpBackupCoreSys.MpLink := ADR(gMpLinkBackupCore);
	MpFileManagerUIBackup.MpLink := ADR(gMpLinkFileManagerUIBackup);
	MpFileManagerUIBackup.UIConnect := ADR(MpFileManagerUIConnect);
	MpBackupCoreConfigSys.MpLink := ADR(gMpLinkBackupCore);
	MpBackupCoreConfigSys.Configuration := ADR(MpBackupConfiguration);

	// Call function blocks
	MpBackupCoreSys();
	MpFileManagerUIBackup();
	MpBackupCoreConfigSys();

END_PROGRAM

PROGRAM _EXIT

	// Disable the function blocks to unlink the MpLinks
	MpBackupCoreSys.Enable := FALSE;
	MpFileManagerUIBackup.Enable := FALSE;
	MpBackupCoreConfigSys.Enable := FALSE;

	// Call function blocks
	MpBackupCoreSys();
	MpFileManagerUIBackup();
	MpBackupCoreConfigSys();

END_PROGRAM
```

#### BackupMgr.typ - Local data types
```iecst
(*Structure types*)

TYPE
	BackupHmiInterfaceType : 	STRUCT  (*HMI interface structure*)
		Commands : BackupHmiCommandsType; (*Structure to hold the commands from the HMI*)
		Parameters : BackupHmiParametersType; (*Structure to hold the parameters for the HMI*)
		Status : BackupHmiStatusType; (*Structure to hold the status information from the HMI*)
	END_STRUCT;
	BackupHmiCommandsType : 	STRUCT  (*Structure to hold the commands from the HMI*)
		Create : BOOL; (*Create a backup*)
		Restore : BOOL; (*Restore a backup*)
		Update : BOOL; (*Install an update*)
		Delete : BOOL; (*Delete a backup*)
		SaveConfig : BOOL; (*Save automatic backup configuration settings*)
		Reset : BOOL; (*Error reset*)
	END_STRUCT;
	BackupHmiParametersType : 	STRUCT  (*Structure to hold the parameters for the HMI*)
		Name : STRING[80] := 'myBackup'; (*Name of the backup*)
		AutomaticBackup : AutomaticBackupType; (*Automatic backup settings*)
	END_STRUCT;
	BackupHmiStatusType : 	STRUCT  (*Structure to hold the status information from the HMI*)
		Busy : BOOL; (*Backup is busy executing an action*)
		Error : BOOL; (*Error flag*)
		CreateAllowed : BOOL; (*Bit to indicate it is allowable to create a backup right now*)
		RestoreAllowed : BOOL; (*Bit to indicate it is allowable to restore a backup right now*)
		BackupCtrlEnabled : BOOL; (*Disable control panel for Backup with in Sim*)
		FileNames : ARRAY[0..49]OF STRING[80]; (*Existing backup file names*)
		TimeStamps : ARRAY[0..49]OF DATE_AND_TIME; (*Time stamps for existing backups*)
		Info : MpBackupProjectInfoRequestType; (*Project information (name, configuration ID, configuration version)*)
		DeviceDataProvider : ARRAY[0..MAX_IDX_FILE_DEV]OF STRING[100]; (*Data provider for file device dropdown on automatic backup configuration pop-up*)
		TableConfig : ARRAY[0..1]OF STRING[120]; (*Table configuration for the list of available backups*)
		SimulationActive : BOOL; (*Flag for if simulation is active*)
		SelectedIndex : USINT; (*Index of the selected backup file*)
		LastSelectedIndex : USINT := 255; (*Index of the last selected backup file*)
		LastSelectedDeviceIndex : UINT; (*Index of the last selected file device. Compared with MpFileManagerUIConnect.DeviceList.SelectedIndex*)
		FileOverMax : BOOL; (*Active when more than 50 items detected*)
		Update : MpBackupAutoUpdateInfoType;
	END_STRUCT;
	AutomaticBackupType : 	STRUCT  (*Automatic backup settings*)
		Enable : BOOL; (*Enable automatic backup feature*)
		Prefix : STRING[50]; (*Name prefix for each automatic backup file*)
		Device : STRING[255]; (*File device to store the automatic backup*)
		Mode : AutomaticBackupModeType; (*Automatic backup time interval*)
		OverwriteOldest : MpBackupOverwriteOldestType; (*Defines whether older backups should be deleted or not*)
	END_STRUCT;
	AutomaticBackupModeType : 	STRUCT  (*Automatic backup time interval*)
		Interval : AutomaticBackupIntervalEnum; (*Day interval (daily, or a specfiic day of the week)*)
		Hour : USINT; (*Time (hour)*)
		Minute : USINT; (*Time (minutes)*)
	END_STRUCT;
END_TYPE

(*Enumerations*)

TYPE
	AutomaticBackupIntervalEnum :
		( (*Selection for how often to automatically create a backup*)
		BACKUP_EVERYDAY, (*Every day*)
		BACKUP_MONDAY, (*Every Monday*)
		BACKUP_TUESDAY, (*Every Tuesday*)
		BACKUP_WEDNESDAY, (*Every Wednesday*)
		BACKUP_THURSDAY, (*Every Thursday*)
		BACKUP_FRIDAY, (*Every Friday*)
		BACKUP_SATURDAY, (*Every Saturday*)
		BACKUP_SUNDAY (*Every Sunday*)
		);
	BackupStateEnum :
		( (*States for backup state machine*)
		BACKUP_IDLE, (*Wait state*)
		BACKUP_CREATING, (*Creating a backup*)
		BACKUP_AUTOCREATE, (*Autobackup in progress*)
		BACKUP_REFRESHING_LIST, (*Refreshing backup list*)
		BACKUP_RESTORING, (*Restoring a backup*)
		BACKUP_UPDATING, (*Installing a new version*)
		BACKUP_DELETING, (*Deleting a backup*)
		BACKUP_SIM, (*CPU in simulation mode, don't do anything*)
		BACKUP_ERROR (*Error state*)
		);
END_TYPE
```

#### BackupMgr.var - Local variables
```iecst
(*Function Blocks*)
VAR
	MpBackupCoreSys : MpBackupCore; (*MpBackupCore instance*)
	MpBackupCoreConfigSys : MpBackupCoreConfig; (*MpBackupCoreConfig instance*)
	MpFileManagerUIBackup : MpFileManagerUI; (*MpFileManagerUI instance*)
	DirCreateBackup : DirCreate; (*DirCreate instance*)
END_VAR
(*Constants*)
VAR CONSTANT
	MAX_IDX_FILE_DEV : USINT := MAX_IDX_USB_DEV_LIST + 1; (*Maximum number of  file devices *)
END_VAR
(*Structure Types*)
VAR
	MpBackupConfiguration : MpBackupCoreConfigType; (*MpBackup configuration*)
	MpFileManagerUIConnect : MpFileManagerUIConnectType; (*MpFile connection to the HMI*)
	HmiBackup : BackupHmiInterfaceType; (*HMI interface structure*)
END_VAR
(*Enumerations*)
VAR
	BackupState : BackupStateEnum; (*States for backup state machine*)
END_VAR
(*Variables*)
VAR
	i : USINT; (*Index for loops*)
	DeviceCount : USINT; (*Counter for available file devices*)
	ItemCount : UDINT;
END_VAR
VAR RETAIN
	AutomaticBackupRetain : AutomaticBackupType;
END_VAR
```

#### HMIActions.st - Supporting code for the HMI interface
```iecst
ACTION FormatDeviceDataProvider:

	// Select CF device if USB device is not available
	FOR i := 0 TO ((SIZEOF(gUSBAvailable) / SIZEOF(gUSBAvailable[0])) - 1) DO
		IF gUSBAvailable[i] THEN
			HmiBackup.Status.DeviceDataProvider[i + 1] := '{"value":"USB';
			brsitoa(i + 1, ADR(HmiBackup.Status.DeviceDataProvider[i + 1]) + brsstrlen(ADR(HmiBackup.Status.DeviceDataProvider[i + 1])));
			brsstrcat(ADR(HmiBackup.Status.DeviceDataProvider[i + 1]), ADR('","text":"USB'));
			brsitoa(i + 1, ADR(HmiBackup.Status.DeviceDataProvider[i + 1]) + brsstrlen(ADR(HmiBackup.Status.DeviceDataProvider[i + 1])));
			brsstrcat(ADR(HmiBackup.Status.DeviceDataProvider[i + 1]), ADR('"}'));
			MpFileManagerUIConnect.DeviceList.DeviceNames[i + 1] := 'USB';
			brsitoa(i + 1, ADR(MpFileManagerUIConnect.DeviceList.DeviceNames[i + 1]) + brsstrlen(ADR(MpFileManagerUIConnect.DeviceList.DeviceNames[i + 1])));
		ELSE
			brsmemset(ADR(HmiBackup.Status.DeviceDataProvider[i + 1]), 0, SIZEOF(HmiBackup.Status.DeviceDataProvider[i + 1]));
			brsmemset(ADR(MpFileManagerUIConnect.DeviceList.DeviceNames[i + 1]), 0, SIZEOF(MpFileManagerUIConnect.DeviceList.DeviceNames[i + 1]));
		END_IF
	END_FOR

	// Configure visible device list
	HmiBackup.Status.TableConfig[0] := '{ "specRows": [{"from":';
	FOR i := 0 TO ((SIZEOF(MpFileManagerUIConnect.DeviceList.DeviceNames)/SIZEOF(MpFileManagerUIConnect.DeviceList.DeviceNames[0])) - 1) DO
		IF MpFileManagerUIConnect.DeviceList.DeviceNames[i] <> '' THEN
			DeviceCount := i + 1;
		END_IF
	END_FOR
	brsitoa((DeviceCount), ADR(HmiBackup.Status.TableConfig[0]) + brsstrlen(ADR(HmiBackup.Status.TableConfig[0])));
	brsstrcat(ADR(HmiBackup.Status.TableConfig[0]), ADR(',"to":9, "visible":false}]}'));

	// Configure visible file list
	ItemCount := MpFileManagerUIConnect.File.PathInfo.FileCount + MpFileManagerUIConnect.File.PathInfo.FolderCount;
	HmiBackup.Status.TableConfig[1] := '{ "specRows": [{"from":';
	brsitoa((ItemCount), ADR(HmiBackup.Status.TableConfig[1]) + brsstrlen(ADR(HmiBackup.Status.TableConfig[1])));
	brsstrcat(ADR(HmiBackup.Status.TableConfig[1]), ADR(',"to":50, "visible":false}]}'));

	HmiBackup.Status.FileOverMax := ItemCount > (SIZEOF(MpFileManagerUIConnect.File.List.Items)/SIZEOF(MpFileManagerUIConnect.File.List.Items[0]));

END_ACTION

ACTION SaveBackupConfiguration:

	MpBackupConfiguration.AutomaticBackup.Enabled := HmiBackup.Parameters.AutomaticBackup.Enable;
	MpBackupConfiguration.AutomaticBackup.NamePrefix := HmiBackup.Parameters.AutomaticBackup.Prefix;
	MpBackupConfiguration.AutomaticBackup.DeviceName := HmiBackup.Parameters.AutomaticBackup.Device;
	MpBackupConfiguration.AutomaticBackup.OverwriteOldest := HmiBackup.Parameters.AutomaticBackup.OverwriteOldest;
	MpBackupConfiguration.AutomaticBackup.Mode.Time := UDINT_TO_TOD((((USINT_TO_UDINT(HmiBackup.Parameters.AutomaticBackup.Mode.Hour) * 60) + HmiBackup.Parameters.AutomaticBackup.Mode.Minute) * 60) * 1000);
	CASE HmiBackup.Parameters.AutomaticBackup.Mode.Interval OF
		BACKUP_EVERYDAY:
			MpBackupConfiguration.AutomaticBackup.Mode.Interval := mpBACKUP_INTERVAL_DAILY;
		BACKUP_MONDAY:
			MpBackupConfiguration.AutomaticBackup.Mode.Interval := mpBACKUP_INTERVAL_WEEKLY;
			MpBackupConfiguration.AutomaticBackup.Mode.Day := mpBACKUP_DAY_MONDAY;
		BACKUP_TUESDAY:
			MpBackupConfiguration.AutomaticBackup.Mode.Interval := mpBACKUP_INTERVAL_WEEKLY;
			MpBackupConfiguration.AutomaticBackup.Mode.Day := mpBACKUP_DAY_TUESDAY;
		BACKUP_WEDNESDAY:
			MpBackupConfiguration.AutomaticBackup.Mode.Interval := mpBACKUP_INTERVAL_WEEKLY;
			MpBackupConfiguration.AutomaticBackup.Mode.Day := mpBACKUP_DAY_WEDNESDAY;
		BACKUP_THURSDAY:
			MpBackupConfiguration.AutomaticBackup.Mode.Interval := mpBACKUP_INTERVAL_WEEKLY;
			MpBackupConfiguration.AutomaticBackup.Mode.Day := mpBACKUP_DAY_THURSDAY;
		BACKUP_FRIDAY:
			MpBackupConfiguration.AutomaticBackup.Mode.Interval := mpBACKUP_INTERVAL_WEEKLY;
			MpBackupConfiguration.AutomaticBackup.Mode.Day := mpBACKUP_DAY_FRIDAY;
		BACKUP_SATURDAY:
			MpBackupConfiguration.AutomaticBackup.Mode.Interval := mpBACKUP_INTERVAL_WEEKLY;
			MpBackupConfiguration.AutomaticBackup.Mode.Day := mpBACKUP_DAY_SATURDAY;
		BACKUP_SUNDAY:
			MpBackupConfiguration.AutomaticBackup.Mode.Interval := mpBACKUP_INTERVAL_WEEKLY;
			MpBackupConfiguration.AutomaticBackup.Mode.Day := mpBACKUP_DAY_SUNDAY;
	END_CASE

	// Save current backup setings to retain variable
	AutomaticBackupRetain := HmiBackup.Parameters.AutomaticBackup;

 END_ACTION

ACTION LoadBackupConfiguration:

	HmiBackup.Parameters.AutomaticBackup.Enable := MpBackupConfiguration.AutomaticBackup.Enabled;
	HmiBackup.Parameters.AutomaticBackup.Prefix := MpBackupConfiguration.AutomaticBackup.NamePrefix;
	HmiBackup.Parameters.AutomaticBackup.Device := MpBackupConfiguration.AutomaticBackup.DeviceName;
	HmiBackup.Parameters.AutomaticBackup.OverwriteOldest := MpBackupConfiguration.AutomaticBackup.OverwriteOldest;
	HmiBackup.Parameters.AutomaticBackup.Mode.Hour := UDINT_TO_USINT(TOD_TO_UDINT(MpBackupConfiguration.AutomaticBackup.Mode.Time) / 1000 / 60 / 60);
	HmiBackup.Parameters.AutomaticBackup.Mode.Minute := UDINT_TO_USINT(TOD_TO_UDINT(MpBackupConfiguration.AutomaticBackup.Mode.Time) / 1000 / 60) - (HmiBackup.Parameters.AutomaticBackup.Mode.Hour * 60);
	CASE MpBackupConfiguration.AutomaticBackup.Mode.Interval OF
		mpBACKUP_INTERVAL_DAILY:
			HmiBackup.Parameters.AutomaticBackup.Mode.Interval := BACKUP_EVERYDAY;
		mpBACKUP_INTERVAL_WEEKLY:
			CASE MpBackupConfiguration.AutomaticBackup.Mode.Day OF
				mpBACKUP_DAY_MONDAY:
					HmiBackup.Parameters.AutomaticBackup.Mode.Interval := BACKUP_MONDAY;
				mpBACKUP_DAY_TUESDAY:
					HmiBackup.Parameters.AutomaticBackup.Mode.Interval := BACKUP_TUESDAY;
				mpBACKUP_DAY_WEDNESDAY:
					HmiBackup.Parameters.AutomaticBackup.Mode.Interval := BACKUP_WEDNESDAY;
				mpBACKUP_DAY_THURSDAY:
					HmiBackup.Parameters.AutomaticBackup.Mode.Interval := BACKUP_THURSDAY;
				mpBACKUP_DAY_FRIDAY:
					HmiBackup.Parameters.AutomaticBackup.Mode.Interval := BACKUP_FRIDAY;
				mpBACKUP_DAY_SATURDAY:
					HmiBackup.Parameters.AutomaticBackup.Mode.Interval := BACKUP_SATURDAY;
				mpBACKUP_DAY_SUNDAY:
					HmiBackup.Parameters.AutomaticBackup.Mode.Interval := BACKUP_SUNDAY;
			END_CASE
	END_CASE
END_ACTION

ACTION FileManager:

	MpFileManagerUIBackup.MpLink := ADR(gMpLinkFileManagerUIBackup);
	MpFileManagerUIBackup.UIConnect := ADR(MpFileManagerUIConnect);
	MpFileManagerUIBackup();
	FOR i := 0 TO ((SIZEOF(HmiBackup.Status.FileNames)/SIZEOF(HmiBackup.Status.FileNames[0])) - 1) DO
		HmiBackup.Status.FileNames[i] := MpFileManagerUIConnect.File.List.Items[i].Name;
		HmiBackup.Status.TimeStamps[i] := MpFileManagerUIConnect.File.List.Items[i].LastModified;
	END_FOR

	IF ((MpFileManagerUIConnect.DeviceList.SelectedIndex <> HmiBackup.Status.LastSelectedDeviceIndex) AND (MpFileManagerUIConnect.Status = mpFILE_UI_STATUS_IDLE)) THEN
		HmiBackup.Status.LastSelectedDeviceIndex := MpFileManagerUIConnect.DeviceList.SelectedIndex;
		IF HmiBackup.Status.LastSelectedIndex >= MpFileManagerUIConnect.File.PathInfo.FolderCount THEN
			HmiBackup.Status.SelectedIndex := 0;
		ELSE
			HmiBackup.Status.LastSelectedIndex := HmiBackup.Status.LastSelectedIndex + 1;
		END_IF
	END_IF

END_ACTION
```

### Package Logical/Infrastructure/File - Package for mapp File Framework

### Program Logical/Infrastructure/File/FileMgr (IEC) - File manager

#### FileMgr.typ
```iecst
(*Structure types*)

TYPE
	FileHmiInterfaceType : 	STRUCT  (*Structure to hold commands, parameters and status from the HMI*)
		Commands : FileHmiCommandsType; (*Structure to hold the commands from the HMI*)
		Parameters : FileHmiParametersType; (*Structure to hold parameters for the mapp View HMI*)
		Status : FileHmiStatusType; (*Structure to hold status information from the mapp View HMI*)
	END_STRUCT;
	FileHmiCommandsType : 	STRUCT  (*Structure to hold the commands from the HMI*)
		Delete : BOOL; (*Delete file*)
		FolderUp : BOOL; (*Move back/up a folder*)
		EnterFolder : BOOL; (*Move forward/down a folder*)
		MultiSelect : BOOL; (*Enables the ability to select multiple files*)
		CheckFolder : BOOL; (*Run the FIFO check to determine if old files should be deleted*)
	END_STRUCT;
	FileHmiParametersType : 	STRUCT  (*Structure to hold parameters for the mapp View HMI*)
		OldSortOrder : MpFileManagerUISortOrderEnum; (*Previous sord order*)
		Fifo : FileHmiParaFifoType; (*Parameters for the FIFO feature (first-in-first-out)*)
	END_STRUCT;
	FileHmiStatusType : 	STRUCT  (*Structure to hold status information from the mapp View HMI*)
		FileNames : ARRAY[0..49]OF STRING[80]; (*List of file names*)
		TimeStamps : ARRAY[0..49]OF DATE_AND_TIME; (*List of time stamps for file names*)
		Type : ARRAY[0..49]OF DINT; (*List of file types*)
		Size : ARRAY[0..49]OF UDINT; (*List of file sizes*)
		DeviceDataProvider : ARRAY[0..MAX_IDX_FILE_DEV]OF STRING[100]; (*Data provider for the file device selector*)
		FifoSelect : ARRAY[0..MAX_IDX_FILE_DEV]OF DINT; (*Indicate FIFO selected file device*)
		DeviceName : STRING[50]; (*File device name*)
		FileName : STRING[255]; (*Fille name*)
		TableConfig : ARRAY[0..1]OF STRING[120]; (*Table configuration for the file explorer (table widget) on the mapp View HMI*)
		IsFolder : BOOL; (*Flag for whether the item is a folder (versus a file)*)
		BackButton : BOOL; (*Flag for whether the back button should be shown*)
		DeleteStep : FileDeleteStepEnum; (*Enumeration for automatic file deletion steps*)
		AutoDeleteSelected : USINT; (*Index for automatic file deletion*)
		FolderSize : REAL; (*Size of currently selected folder*)
		SelectedIndex : USINT; (*Selected index in the file list*)
		FifoConfigEnable : BOOL; (*Disable FIFO access or change confirmation when FIFO is active*)
		DefaultFileSelected : BOOL; (*The default recipe is selected*)
	END_STRUCT;
	FileHmiParaFifoType : 	STRUCT  (*Parameters for the FIFO feature (first-in-first-out)*)
		Enable : BOOL; (*FIFO enable*)
		DeviceName : STRING[50]; (*File device that the FIFO is active on*)
		FifoType : FileFifoTypeEnum; (*Defines the delete behavior of the FIFO*)
		ScanInterval : DINT := 60; (*[minutes]*)
		MaxFileAge : UINT := 365; (*[days] Files older than 1 year will be deleted*)
		MaxFolderSize : REAL := 1000; (*[kB] - Max size of files inside the active folder*)
		MaxNumberOfFiles : UINT := 20; (*Max number of files inside active folder*)
	END_STRUCT;
	FilePathCheckType : 	STRUCT  (*Setup for checking available folders / file devices for FIleManager*)
		Folder : ARRAY[0..9]OF STRING[20]; (*Folder name in user partition*)
		PrgName : ARRAY[0..9]OF STRING[12]; (*Program name for mapp framework components*)
		DeviceList : MpFileManagerUIDeviceListType; (*Device name*)
	END_STRUCT;
END_TYPE

(*Enumerations*)

TYPE
	FileDeleteStepEnum :
		( (*Enumeration for file deletion steps*)
		FILE_DISABLED, (*Disabled*)
		FILE_DELETE_WAIT, (*Wait state*)
		FILE_SCAN_FOLDER_WAIT, (*Wait for check for old files command*)
		FILE_SELECT_DEVICE, (*Switch file device to the configured one *)
		FILE_REFRESH, (*Refreshing the data*)
		FILE_SORT_BY_DATE, (*Sort by date so the oldest files are at the end*)
		FILE_SORT_BY_DATE_WAIT, (*Wait step switching sorting mode*)
		FILE_GO_TO_END, (*Pages down until at the end of the file list*)
		FILE_GO_TO_END_1,
		FILE_CHECK_FOR_FILTER, (*Check which delete filter is active*)
		FILE_SELECT_OLDEST_FILES_0, (*Scan and select all file over the filter setting*)
		FILE_CALC_FOLDER_SIZE, (*Calculate the overall file size in the open folder*)
		FILE_CALC_FOLDER_SCROLL,
		FILE_SELECT_OLDEST_FILES_1, (*Scan and select all file over the filter setting*)
		FILE_DELETE_FILES, (*Set command to delete the selected oldest files*)
		FILE_CONFIRM_DELETE, (*Confirm the file delete*)
		FILE_CONFIRM_DELETE_WAIT, (*Wait for the automatic refresh after file deletion*)
		FILE_RESET_SORT_BY, (*Restore old sort order*)
		FILE_RESET_SORT_BY_WAIT (*Waiting for restore previous sort order*)
		);
	FileFifoTypeEnum :
		( (*Defines the delete behavior of the FIFO*)
		FILE_FIFO_NUM_OF_FILES := 0, (*Delete according to total number of files*)
		FILE_FIFO_SIZE_OF_FOLDER (*Delete according to maximum folder size*)
		);
	FileTypeEnum :
		( (*Defines the type of file in order to update the displayed icon*)
		FOLDER := 0, (*Folder*)
		FILE := 1, (*File*)
		FILE_SELECTED := 2 (*The selected file*)
		);
END_TYPE
```

#### FileMgr.var
```iecst
(*Function Blocks*)
VAR
	MpFileManagerUISys : MpFileManagerUI; (*MpFileManagerUI instance*)
	MpFileManagerUI_FIFO : MpFileManagerUI; (*MpFileManagerUI instance*)
	CheckStatusTrigger : R_TRIG; (*Trigger function block*)
	WaitTimer : TON; (*FIFO handling support*)
	ScanFolderTimer : TON; (*Timer to scan for folder*)
	CurrentIndex : UDINT; (*FIFO handling support deleting more then 50 files*)
	DirReadFolderSize : DirRead; (*FIFO handling support reading current folder size*)
END_VAR
(*Constants*)
VAR CONSTANT
	MAX_IDX_FILE_DEV : USINT := MAX_IDX_USB_DEV_LIST + 7; (*Maximum number of  file devices *)
END_VAR
(*Structure Types*)
VAR
	MpFileManagerUIConnect : MpFileManagerUIConnectType; (*File manager connection to the HMI*)
	MpFileManagerUIConnect_FIFO : {REDUND_UNREPLICABLE} MpFileManagerUIConnectType; (*File manager connection to the HMI*)
	HmiFile : FileHmiInterfaceType; (*HMI interface structure*)
	PathCheck : FilePathCheckType; (*Parameter structure controlling the visible file device based on available folders*)
	DirectoryData : fiDIR_READ_DATA; (*FIFO handling support reading current folder size*)
END_VAR
(*Variables*)
VAR
	i : USINT; (*Index for FOR loops*)
	DeviceCount : USINT; (*Counter for available file devices*)
	Ident : UDINT; (*Ident of a program on target*)
	IdentStatus : UINT; (*Status variable if a program exists on target*)
	FolderDepthCount : USINT; (*Keeps track of the folder depth location to determine whether or not the back button should be shown*)
	USBOffset : USINT; (*Device list offset where to add USB device*)
	MaxDeviceNameIndex : USINT; (*How many devices are configured*)
	TempIdx : USINT; (*FIFO handling support index variable*)
	FileNameArraySize : USINT; (*FIFO handling support size of the array*)
	StartIndex : USINT; (*FIFO handling support *)
	Fifo_Count : USINT; (*FIFO handling support current file count*)
END_VAR
VAR RETAIN
	FifoSettingsRetain : {REDUND_UNREPLICABLE} FileHmiParaFifoType; (*Store FIFO settings in retain memory to be applied after boot*)
END_VAR
VAR
	NextOpenIndex : USINT; (*Index for the next open slot in mpFileManagerUICOnnect device list which populates table*)
END_VAR
```

#### FIFOOperations.st
```iecst
ACTION FIFOOperation:

	CheckStatusTrigger(CLK := (MpFileManagerUIConnect_FIFO.Status = mpFILE_UI_STATUS_CHANGE_DIR) OR
							  (MpFileManagerUIConnect_FIFO.Status = mpFILE_UI_STATUS_CHANGE_DEVICE) OR
							  (MpFileManagerUIConnect_FIFO.Status = mpFILE_UI_STATUS_CREATE));

	IF CheckStatusTrigger.Q OR ScanFolderTimer.Q THEN
		HmiFile.Commands.CheckFolder := HmiFile.Parameters.Fifo.Enable;
	END_IF

	brsmemset(ADR(HmiFile.Status.FifoSelect[0]), 0, SIZEOF(HmiFile.Status.FifoSelect));
	FOR i := 0 TO ((SIZEOF(MpFileManagerUIConnect.DeviceList.DeviceNames)/SIZEOF(MpFileManagerUIConnect.DeviceList.DeviceNames[0])) - 1) DO
		IF (HmiFile.Parameters.Fifo.DeviceName = MpFileManagerUIConnect.DeviceList.DeviceNames[i]) AND HmiFile.Parameters.Fifo.Enable THEN
			HmiFile.Status.FifoSelect[i] := 1;
			EXIT;
		END_IF
	END_FOR

	// Autodelete oldest files based on scanning option
	CASE HmiFile.Status.DeleteStep OF
		FILE_DISABLED:
			IF (HmiFile.Parameters.Fifo.Enable) THEN
				MpFileManagerUI_FIFO.Enable := TRUE;
				HmiFile.Status.DeleteStep := FILE_DELETE_WAIT;
			ELSE
				brsmemset(ADR(HmiFile.Status.FifoSelect[0]), 0, SIZEOF(HmiFile.Status.FifoSelect));
			END_IF

		FILE_DELETE_WAIT:
			IF (HmiFile.Parameters.Fifo.Enable) THEN
				// Wait for check the correct device selection
				ScanFolderTimer.IN := TRUE;
				IF ScanFolderTimer.Q THEN
					ScanFolderTimer.IN := FALSE;
					Fifo_Count := 0;
					HmiFile.Status.DeleteStep := FILE_SCAN_FOLDER_WAIT;
				END_IF
			ELSE
				HmiFile.Status.DeleteStep := FILE_DISABLED;
				ScanFolderTimer.IN := FALSE;
			END_IF

		FILE_SCAN_FOLDER_WAIT:
			// Wait for check for old files command
			IF (HmiFile.Commands.CheckFolder) AND ((MpFileManagerUIConnect_FIFO.Status = mpFILE_UI_STATUS_IDLE) OR (MpFileManagerUIConnect_FIFO.Status = mpFILE_UI_STATUS_ERROR)) THEN
				HmiFile.Commands.CheckFolder := FALSE;
				HmiFile.Status.DeleteStep := FILE_SELECT_DEVICE;
				HmiFile.Parameters.OldSortOrder := MpFileManagerUIConnect_FIFO.File.SortOrder;
			END_IF

		FILE_SELECT_DEVICE:
			//
			FOR i := 0 TO ((SIZEOF(MpFileManagerUIConnect_FIFO.DeviceList.DeviceNames)/SIZEOF(MpFileManagerUIConnect_FIFO.DeviceList.DeviceNames[0])) - 1) DO
				IF HmiFile.Parameters.Fifo.DeviceName = MpFileManagerUIConnect_FIFO.DeviceList.DeviceNames[i] THEN
					MpFileManagerUIConnect_FIFO.DeviceList.SelectedIndex := i;
					EXIT;
				END_IF
			END_FOR
			IF (HmiFile.Parameters.Fifo.DeviceName <> MpFileManagerUIConnect_FIFO.DeviceList.DeviceNames[MpFileManagerUIConnect_FIFO.DeviceList.SelectedIndex]) THEN
				// file device not found
				HmiFile.Status.DeleteStep := FILE_DELETE_WAIT;
			ELSIF (MpFileManagerUIConnect_FIFO.Status = mpFILE_UI_STATUS_IDLE) THEN
				MpFileManagerUIConnect_FIFO.File.Refresh := TRUE;
				HmiFile.Status.DeleteStep := FILE_REFRESH;
			END_IF

		FILE_REFRESH:
			IF ((MpFileManagerUIConnect_FIFO.Status = mpFILE_UI_STATUS_IDLE) AND (NOT MpFileManagerUIConnect_FIFO.File.Refresh)) THEN
				HmiFile.Status.DeleteStep := FILE_SORT_BY_DATE;
			END_IF

		FILE_SORT_BY_DATE:
			// Sort by date so the oldest files are at the end
			IF (MpFileManagerUIConnect_FIFO.File.SortOrder <> mpFILE_SORT_BY_MOD_TIME_DESC) THEN
				MpFileManagerUIConnect_FIFO.File.SortOrder := mpFILE_SORT_BY_MOD_TIME_DESC;
			ELSIF (MpFileManagerUIConnect_FIFO.Status = mpFILE_UI_STATUS_IDLE) THEN
				MpFileManagerUIConnect_FIFO.File.Refresh := TRUE;
				MpFileManagerUI_FIFO();
			END_IF

			IF (MpFileManagerUIConnect_FIFO.Status = mpFILE_UI_STATUS_REFRESH) AND (NOT MpFileManagerUIConnect_FIFO.File.Refresh) THEN
				HmiFile.Status.DeleteStep := FILE_SORT_BY_DATE_WAIT;
			END_IF

		FILE_SORT_BY_DATE_WAIT:
			// Wait for the file manager to complete sorting change
			IF (MpFileManagerUIConnect_FIFO.Status = mpFILE_UI_STATUS_IDLE) THEN
				HmiFile.Status.DeleteStep := FILE_GO_TO_END;
			END_IF

		FILE_GO_TO_END:
			IF (MpFileManagerUIConnect_FIFO.Status = mpFILE_UI_STATUS_IDLE) THEN
				FOR i := 0 TO ((SIZEOF(MpFileManagerUIConnect_FIFO.File.List.Items)/SIZEOF(MpFileManagerUIConnect_FIFO.File.List.Items[0])) - 1) DO
					MpFileManagerUIConnect_FIFO.File.List.Items[i].IsSelected := FALSE;
				END_FOR
				IF (MpFileManagerUIConnect_FIFO.File.PathInfo.FileCount >= (SIZEOF(MpFileManagerUIConnect_FIFO.File.List.Items)/SIZEOF(MpFileManagerUIConnect_FIFO.File.List.Items[0]))) THEN
					// Page down until we get to the end, then start deleting
					IF (MpFileManagerUIConnect_FIFO.File.List.RangeStart <> 0) THEN
						MpFileManagerUIConnect_FIFO.File.List.PageDown := TRUE;
						HmiFile.Status.DeleteStep := FILE_GO_TO_END_1;
					ELSE
						Fifo_Count := 0;
						HmiFile.Status.DeleteStep := FILE_CHECK_FOR_FILTER;
					END_IF
				ELSE
					Fifo_Count := 0;
					HmiFile.Status.DeleteStep := FILE_CHECK_FOR_FILTER;
				END_IF
			END_IF

		FILE_GO_TO_END_1:
			WaitTimer.IN := (NOT MpFileManagerUIConnect_FIFO.File.List.PageDown);
			WaitTimer.PT := T#200ms;
			IF (WaitTimer.Q) THEN
				WaitTimer.IN := FALSE;
				Fifo_Count := Fifo_Count + 1;
				// in case we are stuck trying to get to the last page
				HmiFile.Status.DeleteStep := SEL(Fifo_Count > 10, FILE_GO_TO_END, FILE_DELETE_WAIT);
			END_IF
			WaitTimer();

		FILE_CHECK_FOR_FILTER:
			// Check which delete filter is active
			CASE HmiFile.Parameters.Fifo.FifoType OF
				FILE_FIFO_NUM_OF_FILES:
					HmiFile.Status.DeleteStep := SEL(MpFileManagerUIConnect_FIFO.File.PathInfo.FileCount <= HmiFile.Parameters.Fifo.MaxNumberOfFiles, FILE_SELECT_OLDEST_FILES_0, FILE_DELETE_WAIT);

				FILE_FIFO_SIZE_OF_FOLDER:
					CurrentIndex := 0;
					HmiFile.Status.DeleteStep := FILE_CALC_FOLDER_SIZE;
			END_CASE

		FILE_SELECT_OLDEST_FILES_0:
			// Scan and select all file over the filter setting
			IF (MpFileManagerUIConnect_FIFO.Status = mpFILE_UI_STATUS_IDLE) THEN
				IF MpFileManagerUIConnect_FIFO.File.PathInfo.FileCount > 1 THEN
					MpFileManagerUIConnect_FIFO.File.MultiSelect := TRUE;
				END_IF
				HmiFile.Status.AutoDeleteSelected := 0;
				// start from the first file to delete and select everything after
				// e.g. if there are 100 files and we want to keep 60 files around then we'd start at 60 + 0 MOD 50 = 10 and go to index 49
				FileNameArraySize := SIZEOF(MpFileManagerUIConnect_FIFO.File.List.Items)/SIZEOF(MpFileManagerUIConnect_FIFO.File.List.Items[0]);
				IF (HmiFile.Parameters.Fifo.MaxNumberOfFiles >= FileNameArraySize) THEN
					StartIndex := FileNameArraySize - (UDINT_TO_USINT(MpFileManagerUIConnect_FIFO.File.PathInfo.FileCount - HmiFile.Parameters.Fifo.MaxNumberOfFiles + MpFileManagerUIConnect_FIFO.File.PathInfo.FolderCount) MOD FileNameArraySize);
				ELSE
					StartIndex := UDINT_TO_USINT(HmiFile.Parameters.Fifo.MaxNumberOfFiles + MpFileManagerUIConnect_FIFO.File.PathInfo.FolderCount) MOD FileNameArraySize;
				END_IF
				IF (StartIndex = FileNameArraySize) THEN
					StartIndex := 0;
				END_IF

				IF (StartIndex > 0) THEN
					FOR i := 0 TO (StartIndex - 1) DO
						MpFileManagerUIConnect_FIFO.File.List.Items[i].IsSelected := FALSE;
					END_FOR
				END_IF

				FOR i := StartIndex TO (FileNameArraySize - 1) DO
					MpFileManagerUIConnect_FIFO.File.List.Items[i].IsSelected := FALSE;
					IF (MpFileManagerUIConnect_FIFO.File.List.Items[i].ItemType <> mpFILE_ITEM_TYPE_NONE) AND NOT MpFileManagerUIConnect_FIFO.File.List.Items[i].IsFolder THEN
						MpFileManagerUIConnect_FIFO.File.List.Items[i].IsSelected := TRUE;
						HmiFile.Status.AutoDeleteSelected := HmiFile.Status.AutoDeleteSelected + 1;
					END_IF
				END_FOR

				IF (HmiFile.Status.AutoDeleteSelected > 0) THEN
					HmiFile.Status.DeleteStep := FILE_DELETE_FILES;
				ELSE
					MpFileManagerUIConnect_FIFO.File.MultiSelect := FALSE;
					HmiFile.Status.DeleteStep := FILE_RESET_SORT_BY;
				END_IF
			END_IF

		FILE_CALC_FOLDER_SIZE:
			IF (CurrentIndex = 0) THEN
				HmiFile.Status.FolderSize := 0;
			END_IF
			DirReadFolderSize.enable := TRUE;
			DirReadFolderSize.pDevice := ADR(HmiFile.Parameters.Fifo.DeviceName);
			DirReadFolderSize.pPath := 0;
			DirReadFolderSize.entry := CurrentIndex;
			DirReadFolderSize.option := fiFILE;
			DirReadFolderSize.pData := ADR(DirectoryData);
			DirReadFolderSize.data_len := SIZEOF(DirectoryData);
			DirReadFolderSize();
			IF ((DirReadFolderSize.status = ERR_OK) OR (DirReadFolderSize.status = fiERR_NO_MORE_ENTRIES)) THEN
				HmiFile.Status.FolderSize := HmiFile.Status.FolderSize + UDINT_TO_REAL(DirectoryData.Filelength);
				CurrentIndex := CurrentIndex + 1;
				IF (CurrentIndex >= MpFileManagerUIConnect_FIFO.File.PathInfo.FileCount) THEN
					HmiFile.Status.DeleteStep := SEL(HmiFile.Status.FolderSize > HmiFile.Parameters.Fifo.MaxFolderSize*1024, FILE_RESET_SORT_BY, FILE_SELECT_OLDEST_FILES_1);
				END_IF
			END_IF

		FILE_SELECT_OLDEST_FILES_1:
			// Scan and select all file over the filter setting
			IF (MpFileManagerUIConnect_FIFO.Status = mpFILE_UI_STATUS_IDLE) THEN
				FOR i:=0 TO ((SIZEOF(MpFileManagerUIConnect_FIFO.File.List.Items)/SIZEOF(MpFileManagerUIConnect_FIFO.File.List.Items[0])) - 1) DO
					MpFileManagerUIConnect_FIFO.File.List.Items[i].IsSelected := FALSE;
				END_FOR
				FOR i:=0 TO ((SIZEOF(MpFileManagerUIConnect_FIFO.File.List.Items)/SIZEOF(MpFileManagerUIConnect_FIFO.File.List.Items[0])) - 1) DO
					IF ((MpFileManagerUIConnect_FIFO.File.List.Items[i].Size = 0) OR
						((HmiFile.Parameters.Fifo.MaxFolderSize*1024) > (HmiFile.Status.FolderSize - UDINT_TO_REAL(MpFileManagerUIConnect_FIFO.File.List.Items[i].Size)))) THEN
						EXIT;
					END_IF
					MpFileManagerUIConnect_FIFO.File.List.Items[i].IsSelected := TRUE;
					HmiFile.Status.FolderSize := HmiFile.Status.FolderSize - UDINT_TO_REAL(MpFileManagerUIConnect_FIFO.File.List.Items[i].Size);
				END_FOR
				MpFileManagerUIConnect_FIFO.File.MultiSelect := (i > 1);
				HmiFile.Status.DeleteStep := FILE_DELETE_FILES;
			END_IF

		FILE_DELETE_FILES:
			// Set command to delete the selected oldest files
			IF (MpFileManagerUIConnect_FIFO.Status = mpFILE_UI_STATUS_IDLE) THEN
				MpFileManagerUIConnect_FIFO.File.Delete := TRUE;
			END_IF

			IF (MpFileManagerUIConnect_FIFO.Status = mpFILE_UI_STATUS_DELETE) THEN
				HmiFile.Status.DeleteStep := FILE_CONFIRM_DELETE;
			END_IF

		FILE_CONFIRM_DELETE:
			// Confirm the file delete
			IF (MpFileManagerUIConnect_FIFO.MessageBox.Type = mpFILE_MSG_CONFIRM_DELETE) THEN
				MpFileManagerUIConnect_FIFO.MessageBox.Confirm := TRUE;
			ELSIF (MpFileManagerUIConnect_FIFO.Status = mpFILE_UI_STATUS_IDLE) AND (MpFileManagerUIConnect_FIFO.MessageBox.LayerStatus = 1) THEN
				HmiFile.Status.DeleteStep := FILE_CONFIRM_DELETE_WAIT;
			END_IF

		FILE_CONFIRM_DELETE_WAIT:
			IF ((MpFileManagerUIConnect_FIFO.Status = mpFILE_UI_STATUS_REFRESH) OR (MpFileManagerUIConnect_FIFO.Status = mpFILE_UI_STATUS_IDLE)) THEN
				MpFileManagerUIConnect_FIFO.File.MultiSelect := FALSE;
				IF (HmiFile.Parameters.Fifo.FifoType = FILE_FIFO_SIZE_OF_FOLDER) THEN
					HmiFile.Status.DeleteStep := SEL((HmiFile.Status.FolderSize > (HmiFile.Parameters.Fifo.MaxFolderSize*1024)), FILE_RESET_SORT_BY, FILE_GO_TO_END);
				ELSE
					// if more files need to be deleted then go back to select the oldest files
					HmiFile.Status.DeleteStep := SEL((MpFileManagerUIConnect_FIFO.File.PathInfo.FileCount > HmiFile.Parameters.Fifo.MaxNumberOfFiles), FILE_RESET_SORT_BY, FILE_GO_TO_END);
				END_IF
			END_IF

		FILE_RESET_SORT_BY:
			// Restore old sort order
			IF (MpFileManagerUIConnect_FIFO.File.SortOrder <> HmiFile.Parameters.OldSortOrder) THEN
				MpFileManagerUIConnect_FIFO.File.SortOrder := HmiFile.Parameters.OldSortOrder;
			ELSIF (MpFileManagerUIConnect_FIFO.Status = mpFILE_UI_STATUS_IDLE) THEN
				MpFileManagerUIConnect_FIFO.File.Refresh := TRUE;
				HmiFile.Status.DeleteStep := FILE_RESET_SORT_BY_WAIT;
			END_IF

		FILE_RESET_SORT_BY_WAIT:
			// Wait for file manager to complete restoring previous sorting mode
			IF (MpFileManagerUIConnect_FIFO.Status = mpFILE_UI_STATUS_REFRESH) OR (MpFileManagerUIConnect_FIFO.Status = mpFILE_UI_STATUS_IDLE) THEN
				HmiFile.Status.DeleteStep := FILE_DELETE_WAIT;
				IF (MpFileManagerUIConnect_FIFO.MessageBox.Type = mpFILE_MSG_BUSY) THEN
					MpFileManagerUIConnect_FIFO.MessageBox.Confirm := TRUE;
				END_IF
			END_IF
	END_CASE

	// Save current archive setings to retain variable
	FifoSettingsRetain := HmiFile.Parameters.Fifo;

	// Timer to scan file device in intervals
	ScanFolderTimer(PT := DINT_TO_TIME(HmiFile.Parameters.Fifo.ScanInterval * 60000));

	MpFileManagerUIConnect_FIFO.DeviceList.DeviceNames[0] := HmiFile.Parameters.Fifo.DeviceName;
	MpFileManagerUI_FIFO.UIConnect := ADR(MpFileManagerUIConnect_FIFO);
	MpFileManagerUI_FIFO.UISetup.FileListSize := SIZEOF(MpFileManagerUIConnect_FIFO.File.List.Items) / SIZEOF(MpFileManagerUIConnect_FIFO.File.List.Items[0]);

END_ACTION
```
